KUKA KRL program: MyProgram_342().src

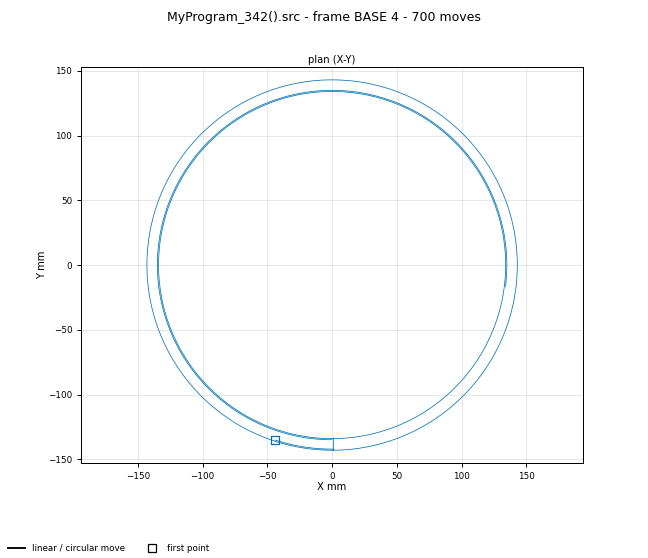
[picture p0: tool path of MyProgram_342().src in frame BASE 4, 700 of 700 moves have a stored position in this frame; points joined in program order, loops and branches not executed]
&ACCESS RVP
&REL 1
&PARAM TEMPLATE = C:\KRC\Roboter\Template\vorgabe
&PARAM EDITMASK = *
DEF MyProgram_342()
; ---- Setting reference (Base) ----
$BASE = BASE_DATA[4]

; --------------------------
; ---- Setting tool (TCP) ----
$TOOL = TOOL_DATA[3]
; --------------------------

$VEL.CP = VEL_APROX_PRINT
Startdeposition()
$VEL.CP = VEL_PRINT
LIN {X -44.0443,Y -135.0812,Z 191,A -94.9972,B 0.9183,C 0.2037,E1 0.9053,E2 187.7978} C_DIS
LIN {X -40.4187,Y -136.2083,Z 191,A -93.5168,B 0.9182,C 0.2043,E1 0.9093,E2 186.3246} C_DIS
LIN {X -37.0832,Y -137.1539,Z 191,A -92.1234,B 0.9181,C 0.2047,E1 0.9131,E2 184.9314} C_DIS
LIN {X -34.1943,Y -137.9034,Z 191,A -90.8718,B 0.9181,C 0.2049,E1 0.9166,E2 183.672} C_DIS
LIN {X -30.5962,Y -138.7458,Z 191,A -89.5644,B 0.9179,C 0.2055,E1 0.9201,E2 182.392} C_DIS
LIN {X -27.1259,Y -139.4652,Z 191,A -87.9953,B 0.9179,C 0.2052,E1 0.9245,E2 180.801} C_DIS
LIN {X -23.7617,Y -140.0774,Z 191,A -86.7669,B 0.9179,C 0.2056,E1 0.9279,E2 179.5949} C_DIS
LIN {X -20.9391,Y -140.5289,Z 191,A -85.3937,B 0.918,C 0.205,E1 0.9318,E2 178.1876} C_DIS
LIN {X -16.902,Y -141.0692,Z 191,A -84.0993,B 0.9178,C 0.2057,E1 0.9353,E2 176.9455} C_DIS
LIN {X -14.3962,Y -141.3492,Z 191,A -82.7514,B 0.9181,C 0.2046,E1 0.9393,E2 175.5466} C_DIS
LIN {X -10.0552,Y -141.7222,Z 191,A -81.1558,B 0.9181,C 0.2046,E1 0.9437,E2 173.9748} C_DIS
LIN {X -6.754,Y -141.9181,Z 191,A -79.8698,B 0.9181,C 0.2043,E1 0.9473,E2 172.6955} C_DIS
LIN {X -3.1252,Y -142.0459,Z 191,A -78.3714,B 0.9183,C 0.2036,E1 0.9516,E2 171.191} C_DIS
LIN {X 0.5232,Y -142.0775,Z 191,A -76.8992,B 0.9185,C 0.2029,E1 0.9557,E2 169.7179} C_DIS
LIN {X 0.5232,Y -142.0775,Z 191,A -76.8992,B 0.9185,C 0.2029,E1 0.9557,E2 169.7179} C_DIS
Enddeposition()
LIN {X 1.0243,Y -142.9726,Z 191,A -77.066,B 0.9181,C 0.2043,E1 0.955,E2 169.9648} C_DIS
Startdeposition()
$VEL.CP = VEL_PRINT
LIN {X -1.7511,Y -142.9678,Z 191,A -78.3434,B 0.9179,C 0.2053,E1 0.9513,E2 171.2682} C_DIS
LIN {X -5.1484,Y -142.885,Z 191,A -79.7715,B 0.9177,C 0.2061,E1 0.9473,E2 172.7072} C_DIS
LIN {X -8.6494,Y -142.7153,Z 191,A -81.1441,B 0.9177,C 0.2064,E1 0.9434,E2 174.0755} C_DIS
LIN {X -12.1449,Y -142.4604,Z 191,A -82.5233,B 0.9176,C 0.2067,E1 0.9395,E2 175.4516} C_DIS
LIN {X -15.6335,Y -142.1201,Z 191,A -83.9093,B 0.9176,C 0.2069,E1 0.9356,E2 176.8354} C_DIS
LIN {X -19.1308,Y -141.6924,Z 191,A -85.3144,B 0.9175,C 0.2071,E1 0.9316,E2 178.2402} C_DIS
LIN {X -22.712,Y -141.1639,Z 191,A -86.7484,B 0.9175,C 0.2071,E1 0.9276,E2 179.6723} C_DIS
LIN {X -25.7644,Y -140.6376,Z 191,A -88.0735,B 0.9175,C 0.2073,E1 0.9239,E2 181.0107} C_DIS
LIN {X -29.4674,Y -139.9092,Z 191,A -89.5418,B 0.9175,C 0.2071,E1 0.9198,E2 182.4729} C_DIS
LIN {X -33.0283,Y -139.1105,Z 191,A -90.9656,B 0.9175,C 0.2068,E1 0.9159,E2 183.8914} C_DIS
LIN {X -36.4402,Y -138.2557,Z 191,A -92.3295,B 0.9177,C 0.2064,E1 0.9122,E2 185.2488} C_DIS
LIN {X -39.8092,Y -137.3234,Z 191,A -93.8498,B 0.9177,C 0.2063,E1 0.908,E2 186.7878} C_DIS
LIN {X -43.0482,Y -136.343,Z 191,A -95.202,B 0.9177,C 0.2058,E1 0.9043,E2 188.14} C_DIS
LIN {X -46.4782,Y -135.2119,Z 191,A -96.7128,B 0.9179,C 0.2053,E1 0.9003,E2 189.6609} C_DIS
LIN {X -49.0096,Y -134.3156,Z 191,A -97.9561,B 0.9179,C 0.2051,E1 0.8969,E2 190.9301} C_DIS
LIN {X -53.0946,Y -132.7533,Z 191,A -99.6242,B 0.9182,C 0.2039,E1 0.8925,E2 192.5858} C_DIS
LIN {X -56.2262,Y -131.4582,Z 191,A -101.0289,B 0.9184,C 0.2032,E1 0.8888,E2 193.998} C_DIS
LIN {X -58.6861,Y -130.3778,Z 191,A -102.1543,B 0.9185,C 0.2025,E1 0.8859,E2 195.131} C_DIS
LIN {X -61.8637,Y -128.9001,Z 191,A -103.6197,B 0.9187,C 0.2015,E1 0.8821,E2 196.6061} C_DIS
LIN {X -65.0103,Y -127.342,Z 191,A -105.099,B 0.919,C 0.2005,E1 0.8783,E2 198.0966} C_DIS
LIN {X -68.3884,Y -125.5624,Z 191,A -106.7802,B 0.9192,C 0.1993,E1 0.8741,E2 199.8012} C_DIS
LIN {X -72.0014,Y -123.5268,Z 191,A -108.4575,B 0.9196,C 0.1977,E1 0.87,E2 201.481} C_DIS
LIN {X -74.9587,Y -121.7544,Z 191,A -109.9364,B 0.9198,C 0.1964,E1 0.8664,E2 202.9748} C_DIS
LIN {X -78.5539,Y -119.4662,Z 191,A -111.7694,B 0.9202,C 0.1947,E1 0.862,E2 204.8271} C_DIS
LIN {X -82.1648,Y -117.0125,Z 191,A -113.6368,B 0.9206,C 0.1927,E1 0.8576,E2 206.7124} C_DIS
LIN {X -85.116,Y -114.8837,Z 191,A -115.2771,B 0.921,C 0.191,E1 0.8538,E2 208.3803} C_DIS
LIN {X -88.608,Y -112.2125,Z 191,A -117.0907,B 0.9215,C 0.1887,E1 0.8497,E2 210.2018} C_DIS
LIN {X -91.5174,Y -109.8528,Z 191,A -118.854,B 0.9219,C 0.1867,E1 0.8458,E2 212.0045} C_DIS
LIN {X -94.7125,Y -107.1094,Z 191,A -120.5293,B 0.9224,C 0.1842,E1 0.8422,E2 213.6779} C_DIS
LIN {X -97.2632,Y -104.7989,Z 191,A -122.0448,B 0.9228,C 0.1821,E1 0.839,E2 215.2137} C_DIS
LIN {X -99.8004,Y -102.3863,Z 191,A -123.6022,B 0.9232,C 0.1799,E1 0.8358,E2 216.7943} C_DIS
LIN {X -102.7691,Y -99.4052,Z 191,A -125.495,B 0.9237,C 0.1771,E1 0.832,E2 218.7178} C_DIS
LIN {X -105.3467,Y -96.6693,Z 191,A -127.1186,B 0.9242,C 0.1745,E1 0.8289,E2 220.3587} C_DIS
LIN {X -108.0416,Y -93.6488,Z 191,A -128.8309,B 0.9248,C 0.1716,E1 0.8257,E2 222.0841} C_DIS
LIN {X -110.0019,Y -91.3373,Z 191,A -130.4103,B 0.9252,C 0.1694,E1 0.8227,E2 223.7174} C_DIS
LIN {X -112.7081,Y -87.977,Z 191,A -132.2096,B 0.9258,C 0.166,E1 0.8195,E2 225.5268} C_DIS
LIN {X -114.8262,Y -85.1932,Z 191,A -133.7873,B 0.9263,C 0.1632,E1 0.8168,E2 227.1302} C_DIS
LIN {X -116.9319,Y -82.2791,Z 191,A -135.5615,B 0.9268,C 0.1603,E1 0.8139,E2 228.9531} C_DIS
LIN {X -119.3971,Y -78.6588,Z 191,A -137.5331,B 0.9275,C 0.1565,E1 0.8107,E2 230.9559} C_DIS
LIN {X -121.6959,Y -75.054,Z 191,A -139.3334,B 0.9281,C 0.1528,E1 0.808,E2 232.7685} C_DIS
LIN {X -123.5289,Y -71.9976,Z 191,A -140.96,B 0.9286,C 0.1496,E1 0.8057,E2 234.4237} C_DIS
LIN {X -125.2281,Y -68.9993,Z 191,A -142.5485,B 0.9291,C 0.1464,E1 0.8034,E2 236.0418} C_DIS
LIN {X -126.8799,Y -65.9105,Z 191,A -144.1657,B 0.9296,C 0.143,E1 0.8013,E2 237.6895} C_DIS
LIN {X -128.4908,Y -62.7119,Z 191,A -145.7864,B 0.9302,C 0.1396,E1 0.7992,E2 239.3365} C_DIS
LIN {X -129.9345,Y -59.6614,Z 191,A -147.3777,B 0.9307,C 0.1362,E1 0.7973,E2 240.9617} C_DIS
LIN {X -131.3976,Y -56.3662,Z 191,A -148.9997,B 0.9312,C 0.1326,E1 0.7955,E2 242.6086} C_DIS
LIN {X -132.7118,Y -53.1975,Z 191,A -150.6229,B 0.9317,C 0.129,E1 0.7937,E2 244.2667} C_DIS
LIN {X -133.9822,Y -49.9116,Z 191,A -152.2574,B 0.9322,C 0.1254,E1 0.792,E2 245.9323} C_DIS
LIN {X -135.1575,Y -46.6351,Z 191,A -153.8995,B 0.9327,C 0.1216,E1 0.7905,E2 247.609} C_DIS
LIN {X -136.3021,Y -43.1765,Z 191,A -155.5832,B 0.9332,C 0.1177,E1 0.789,E2 249.3237} C_DIS
LIN {X -137.2869,Y -39.934,Z 191,A -157.1687,B 0.9336,C 0.114,E1 0.7877,E2 250.9407} C_DIS
LIN {X -138.2248,Y -36.5561,Z 191,A -158.8107,B 0.9341,C 0.1101,E1 0.7865,E2 252.6153} C_DIS
LIN {X -139.0565,Y -33.2525,Z 191,A -160.4242,B 0.9346,C 0.1063,E1 0.7854,E2 254.2629} C_DIS
LIN {X -139.7677,Y -30.1225,Z 191,A -161.9849,B 0.935,C 0.1026,E1 0.7844,E2 255.8611} C_DIS
LIN {X -140.5458,Y -26.2607,Z 191,A -163.7723,B 0.9354,C 0.0982,E1 0.7835,E2 257.6767} C_DIS
LIN {X -141.1657,Y -22.7011,Z 191,A -165.4595,B 0.9359,C 0.094,E1 0.7827,E2 259.3961} C_DIS
LIN {X -141.663,Y -19.355,Z 191,A -167.1313,B 0.9363,C 0.09,E1 0.782,E2 261.1107} C_DIS
LIN {X -142.1054,Y -15.7707,Z 191,A -168.7912,B 0.9367,C 0.0858,E1 0.7814,E2 262.7989} C_DIS
LIN {X -142.4479,Y -12.292,Z 191,A -170.4387,B 0.937,C 0.0817,E1 0.781,E2 264.4792} C_DIS
LIN {X -142.7058,Y -8.8037,Z 191,A -172.087,B 0.9374,C 0.0776,E1 0.7807,E2 266.1602} C_DIS
LIN {X -142.8807,Y -5.2595,Z 191,A -173.7528,B 0.9377,C 0.0734,E1 0.7805,E2 267.8582} C_DIS
LIN {X -142.9677,Y -1.7607,Z 191,A -175.3545,B 0.938,C 0.0693,E1 0.7804,E2 269.4859} C_DIS
LIN {X -142.9703,Y 1.6027,Z 191,A -177.0572,B 0.9383,C 0.0652,E1 0.7804,E2 271.2353} C_DIS
LIN {X -142.8852,Y 5.1432,Z 191,A -178.7056,B 0.9386,C 0.061,E1 0.7806,E2 272.9134} C_DIS
LIN {X -142.7147,Y 8.659,Z 191,A 179.6384,B 0.9389,C 0.0568,E1 0.7808,E2 274.601} C_DIS
LIN {X -142.46,Y 12.1493,Z 191,A 177.9898,B 0.9391,C 0.0527,E1 0.7812,E2 276.2813} C_DIS
LIN {X -142.1202,Y 15.6329,Z 191,A 176.3393,B 0.9393,C 0.0485,E1 0.7817,E2 277.9634} C_DIS
LIN {X -141.6952,Y 19.1092,Z 191,A 174.6795,B 0.9395,C 0.0444,E1 0.7823,E2 279.6559} C_DIS
LIN {X -141.1673,Y 22.6907,Z 191,A 172.9828,B 0.9397,C 0.0402,E1 0.783,E2 281.3838} C_DIS
LIN {X -140.6491,Y 25.7,Z 191,A 171.4402,B 0.9399,C 0.0365,E1 0.7838,E2 282.9668} C_DIS
LIN {X -139.885,Y 29.5794,Z 191,A 169.6984,B 0.94,C 0.0321,E1 0.7848,E2 284.728} C_DIS
LIN {X -139.1218,Y 32.9815,Z 191,A 168.0174,B 0.9402,C 0.028,E1 0.7858,E2 286.4445} C_DIS
LIN {X -138.2739,Y 36.3721,Z 191,A 166.375,B 0.9402,C 0.0241,E1 0.787,E2 288.1168} C_DIS
LIN {X -137.3203,Y 39.8199,Z 191,A 164.6972,B 0.9404,C 0.02,E1 0.7883,E2 289.8246} C_DIS
LIN {X -136.3377,Y 43.0651,Z 191,A 163.1033,B 0.9404,C 0.0163,E1 0.7896,E2 291.4473} C_DIS
LIN {X -135.1967,Y 46.5221,Z 191,A 161.409,B 0.9404,C 0.0123,E1 0.7912,E2 293.1703} C_DIS
LIN {X -134.0172,Y 49.818,Z 191,A 159.8681,B 0.9405,C 0.0086,E1 0.7927,E2 294.7277} C_DIS
LIN {X -132.7576,Y 53.084,Z 191,A 158.1472,B 0.9405,C 0.0048,E1 0.7945,E2 296.4873} C_DIS
LIN {X -131.2219,Y 56.7725,Z 191,A 156.2286,B 0.9405,C 0.0005,E1 0.7966,E2 298.444} C_DIS
LIN {X -129.6557,Y 60.2643,Z 191,A 154.5046,B 0.9405,C -0.0034,E1 0.7986,E2 300.1906} C_DIS
LIN {X -127.8296,Y 64.0521,Z 191,A 152.5628,B 0.9405,C -0.0076,E1 0.8011,E2 302.1629} C_DIS
LIN {X -126.0944,Y 67.4031,Z 191,A 150.8798,B 0.9405,C -0.0113,E1 0.8033,E2 303.8657} C_DIS
LIN {X -124.3943,Y 70.4918,Z 191,A 149.217,B 0.9405,C -0.0147,E1 0.8056,E2 305.5579} C_DIS
LIN {X -122.6024,Y 73.5643,Z 191,A 147.4166,B 0.9405,C -0.0181,E1 0.8082,E2 307.4027} C_DIS
LIN {X -120.326,Y 77.2305,Z 191,A 145.6237,B 0.9403,C -0.022,E1 0.8109,E2 309.2021} C_DIS
LIN {X -118.3683,Y 80.1987,Z 191,A 143.8437,B 0.9403,C -0.0252,E1 0.8138,E2 311.0236} C_DIS
LIN {X -115.9267,Y 83.6896,Z 191,A 142.0724,B 0.9401,C -0.0288,E1 0.8167,E2 312.8014} C_DIS
LIN {X -113.8414,Y 86.5056,Z 191,A 140.4645,B 0.9401,C -0.0318,E1 0.8194,E2 314.4326} C_DIS
LIN {X -111.5941,Y 89.3859,Z 191,A 138.6711,B 0.9399,C -0.0348,E1 0.8226,E2 316.2639} C_DIS
LIN {X -108.8784,Y 92.6735,Z 191,A 136.9142,B 0.9399,C -0.0381,E1 0.8258,E2 318.0253} C_DIS
LIN {X -106.5362,Y 95.3567,Z 191,A 135.2388,B 0.9397,C -0.0408,E1 0.829,E2 319.7288} C_DIS
LIN {X -103.5904,Y 98.5495,Z 191,A 133.4117,B 0.9396,C -0.0439,E1 0.8325,E2 321.5649} C_DIS
LIN {X -101.103,Y 101.1002,Z 191,A 131.6927,B 0.9394,C -0.0463,E1 0.836,E2 323.3169} C_DIS
LIN {X -97.9581,Y 104.1496,Z 191,A 129.8889,B 0.9393,C -0.0492,E1 0.8397,E2 325.1251} C_DIS
LIN {X -95.3755,Y 106.5195,Z 191,A 128.362,B 0.9392,C -0.0515,E1 0.8429,E2 326.6653} C_DIS
LIN {X -92.7655,Y 108.8002,Z 191,A 126.8125,B 0.9391,C -0.0536,E1 0.8462,E2 328.2323} C_DIS
LIN {X -89.3893,Y 111.5913,Z 191,A 124.9162,B 0.9389,C -0.0561,E1 0.8504,E2 330.1438} C_DIS
LIN {X -86.6273,Y 113.7483,Z 191,A 123.3944,B 0.9388,C -0.058,E1 0.8538,E2 331.6782} C_DIS
LIN {X -83.7666,Y 115.8709,Z 191,A 121.8524,B 0.9387,C -0.0598,E1 0.8574,E2 333.2323} C_DIS
LIN {X -80.2081,Y 118.3619,Z 191,A 120.0024,B 0.9385,C -0.0619,E1 0.8617,E2 335.0937} C_DIS
LIN {X -77.2858,Y 120.2907,Z 191,A 118.4769,B 0.9385,C -0.0634,E1 0.8654,E2 336.6323} C_DIS
LIN {X -73.5668,Y 122.6009,Z 191,A 116.6243,B 0.9383,C -0.0653,E1 0.8699,E2 338.4949} C_DIS
LIN {X -70.5413,Y 124.3661,Z 191,A 115.1433,B 0.9383,C -0.0666,E1 0.8735,E2 339.9839} C_DIS
LIN {X -67.4728,Y 126.0569,Z 191,A 113.6366,B 0.9381,C -0.0679,E1 0.8773,E2 341.5014} C_DIS
LIN {X -64.275,Y 127.7163,Z 191,A 112.1606,B 0.9381,C -0.0691,E1 0.881,E2 342.9801} C_DIS
LIN {X -61.0358,Y 129.2957,Z 191,A 110.5945,B 0.938,C -0.0701,E1 0.885,E2 344.5592} C_DIS
LIN {X -57.9783,Y 130.6944,Z 191,A 109.2192,B 0.9379,C -0.0711,E1 0.8886,E2 345.9368} C_DIS
LIN {X -53.9096,Y 132.4247,Z 191,A 107.2414,B 0.9379,C -0.072,E1 0.8938,E2 347.9367} C_DIS
LIN {X -49.8217,Y 134.0159,Z 191,A 105.5972,B 0.9377,C -0.0731,E1 0.8981,E2 349.5673} C_DIS
LIN {X -46.631,Y 135.1589,Z 191,A 104.1885,B 0.9377,C -0.0737,E1 0.9019,E2 350.981} C_DIS
LIN {X -43.0836,Y 136.3318,Z 191,A 102.5157,B 0.9377,C -0.0741,E1 0.9065,E2 352.6725} C_DIS
LIN {X -38.2252,Y 137.7725,Z 191,A 100.5903,B 0.9376,C -0.0749,E1 0.9117,E2 354.5852} C_DIS
LIN {X -34.3164,Y 138.8,Z 191,A 98.8052,B 0.9376,C -0.075,E1 0.9166,E2 356.388} C_DIS
LIN {X -30.2002,Y 139.751,Z 191,A 97.1875,B 0.9376,C -0.0754,E1 0.9211,E2 357.9965} C_DIS
LIN {X -26.2866,Y 140.5409,Z 191,A 95.6367,B 0.9376,C -0.0756,E1 0.9254,E2 359.5411} C_DIS
LIN {X -22.7225,Y 141.1622,Z 191,A 94.1997,B 0.9376,C -0.0756,E1 0.9294,E2 360.9762} C_DIS
LIN {X -19.3708,Y 141.661,Z 191,A 92.7853,B 0.9376,C -0.0754,E1 0.9334,E2 362.3962} C_DIS
LIN {X -15.7841,Y 142.1039,Z 191,A 91.5335,B 0.9376,C -0.0756,E1 0.9368,E2 363.6255} C_DIS
LIN {X -12.2682,Y 142.4499,Z 191,A 89.9925,B 0.9376,C -0.075,E1 0.9412,E2 365.1799} C_DIS
LIN {X -8.7735,Y 142.7077,Z 191,A 88.6162,B 0.9376,C -0.0747,E1 0.9451,E2 366.5524} C_DIS
LIN {X -5.6927,Y 142.8638,Z 191,A 87.3417,B 0.9376,C -0.0742,E1 0.9487,E2 367.8307} C_DIS
LIN {X -1.7582,Y 142.9677,Z 191,A 85.8854,B 0.9376,C -0.0738,E1 0.9528,E2 369.273} C_DIS
LIN {X 1.7562,Y 142.9677,Z 191,A 84.4997,B 0.9377,C -0.0732,E1 0.9567,E2 370.6556} C_DIS
LIN {X 5.1446,Y 142.8852,Z 191,A 83.1564,B 0.9377,C -0.0725,E1 0.9605,E2 371.9968} C_DIS
LIN {X 8.6439,Y 142.7156,Z 191,A 81.8057,B 0.9378,C -0.0717,E1 0.9643,E2 373.341} C_DIS
LIN {X 12.1399,Y 142.4608,Z 191,A 80.4574,B 0.9378,C -0.0709,E1 0.9681,E2 374.6825} C_DIS
LIN {X 15.4004,Y 142.1452,Z 191,A 79.1661,B 0.938,C -0.07,E1 0.9717,E2 375.9709} C_DIS
LIN {X 19.1264,Y 141.693,Z 191,A 77.756,B 0.938,C -0.0691,E1 0.9756,E2 377.3701} C_DIS
LIN {X 22.3424,Y 141.2213,Z 191,A 76.4997,B 0.9381,C -0.0681,E1 0.9791,E2 378.6208} C_DIS
LIN {X 26.0479,Y 140.5865,Z 191,A 75.0289,B 0.9382,C -0.0668,E1 0.9832,E2 380.0872} C_DIS
LIN {X 29.6046,Y 139.8795,Z 191,A 73.7235,B 0.9382,C -0.0658,E1 0.9868,E2 381.3754} C_DIS
LIN {X 33.0376,Y 139.1083,Z 191,A 72.3827,B 0.9384,C -0.0645,E1 0.9905,E2 382.708} C_DIS
LIN {X 36.4272,Y 138.2592,Z 191,A 71.0407,B 0.9384,C -0.0631,E1 0.9941,E2 384.043} C_DIS
LIN {X 39.7961,Y 137.3273,Z 191,A 69.7337,B 0.9385,C -0.0617,E1 0.9977,E2 385.3391} C_DIS
LIN {X 43.0376,Y 136.3464,Z 191,A 68.4532,B 0.9386,C -0.0603,E1 1.0011,E2 386.6106} C_DIS
LIN {X 45.7652,Y 135.4558,Z 191,A 67.2302,B 0.9387,C -0.0586,E1 1.0044,E2 387.8417} C_DIS
LIN {X 49.8206,Y 134.0163,Z 191,A 65.801,B 0.9388,C -0.0573,E1 1.0081,E2 389.2368} C_DIS
LIN {X 53.0912,Y 132.7546,Z 191,A 64.4671,B 0.9389,C -0.0556,E1 1.0116,E2 390.5623} C_DIS
LIN {X 56.2234,Y 131.4594,Z 191,A 63.2099,B 0.939,C -0.0539,E1 1.0148,E2 391.8077} C_DIS
LIN {X 59.481,Y 130.0179,Z 191,A 61.8734,B 0.9391,C -0.0521,E1 1.0182,E2 393.1335} C_DIS
LIN {X 62.7074,Y 128.493,Z 191,A 60.5917,B 0.9392,C -0.0504,E1 1.0214,E2 394.3979} C_DIS
LIN {X 65.785,Y 126.9458,Z 191,A 59.3322,B 0.9393,C -0.0486,E1 1.0246,E2 395.6431} C_DIS
LIN {X 68.8971,Y 125.2847,Z 191,A 57.993,B 0.9394,C -0.0466,E1 1.0279,E2 396.9736} C_DIS
LIN {X 72.5064,Y 123.2304,Z 191,A 56.3957,B 0.9395,C -0.0439,E1 1.0317,E2 398.5629} C_DIS
LIN {X 76.0974,Y 121.046,Z 191,A 54.8634,B 0.9397,C -0.0415,E1 1.0354,E2 400.0774} C_DIS
LIN {X 79.4847,Y 118.849,Z 191,A 53.3483,B 0.9397,C -0.039,E1 1.0389,E2 401.5803} C_DIS
LIN {X 83.0062,Y 116.4169,Z 191,A 51.9221,B 0.9399,C -0.0369,E1 1.0421,E2 402.9724} C_DIS
LIN {X 85.8738,Y 114.3183,Z 191,A 50.5144,B 0.9399,C -0.0342,E1 1.0453,E2 404.3782} C_DIS
LIN {X 89.3933,Y 111.5881,Z 191,A 48.8798,B 0.9401,C -0.0313,E1 1.0489,E2 405.995} C_DIS
LIN {X 93.1207,Y 108.4964,Z 191,A 47.2025,B 0.9401,C -0.0284,E1 1.0524,E2 407.641} C_DIS
LIN {X 96.5087,Y 105.4944,Z 191,A 45.607,B 0.9402,C -0.0255,E1 1.0557,E2 409.2104} C_DIS
LIN {X 99.1712,Y 102.9957,Z 191,A 44.2678,B 0.9402,C -0.0229,E1 1.0584,E2 410.5349} C_DIS
LIN {X 102.293,Y 99.8955,Z 191,A 42.7319,B 0.9404,C -0.0201,E1 1.0614,E2 412.0435} C_DIS
LIN {X 104.7507,Y 97.3149,Z 191,A 41.4555,B 0.9404,C -0.0176,E1 1.0638,E2 413.3016} C_DIS
LIN {X 107.6524,Y 94.0949,Z 191,A 39.922,B 0.9404,C -0.0145,E1 1.0666,E2 414.8105} C_DIS
LIN {X 109.9618,Y 91.3857,Z 191,A 38.6546,B 0.9405,C -0.012,E1 1.0689,E2 416.0588} C_DIS
LIN {X 112.1609,Y 88.6737,Z 191,A 37.4046,B 0.9405,C -0.0094,E1 1.071,E2 417.2906} C_DIS
LIN {X 114.4124,Y 85.7489,Z 191,A 35.9709,B 0.9405,C -0.0061,E1 1.0734,E2 418.7191} C_DIS
LIN {X 116.9333,Y 82.2771,Z 191,A 34.4626,B 0.9405,C -0.0029,E1 1.0759,E2 420.2017} C_DIS
LIN {X 119.3312,Y 78.7589,Z 191,A 33.0648,B 0.9405,C -0.0002,E1 1.078,E2 421.5616} C_DIS
LIN {X 121.2326,Y 75.8,Z 191,A 31.8082,B 0.9405,C 0.0025,E1 1.0798,E2 422.7994} C_DIS
LIN {X 123.0551,Y 72.8047,Z 191,A 30.5734,B 0.9405,C 0.0052,E1 1.0816,E2 424.0133} C_DIS
LIN {X 124.8026,Y 69.766,Z 191,A 29.2985,B 0.9405,C 0.0082,E1 1.0833,E2 425.2723} C_DIS
LIN {X 126.8917,Y 65.888,Z 191,A 27.7776,B 0.9405,C 0.0115,E1 1.0853,E2 426.7628} C_DIS
LIN {X 128.4917,Y 62.7099,Z 191,A 26.5378,B 0.9405,C 0.0142,E1 1.0868,E2 427.9796} C_DIS
LIN {X 129.9877,Y 59.5464,Z 191,A 25.2979,B 0.9405,C 0.0171,E1 1.0882,E2 429.1993} C_DIS
LIN {X 131.4128,Y 56.3311,Z 191,A 24.0622,B 0.9404,C 0.0199,E1 1.0896,E2 430.4133} C_DIS
LIN {X 132.7108,Y 53.2,Z 191,A 22.8726,B 0.9404,C 0.0227,E1 1.0908,E2 431.5818} C_DIS
LIN {X 134.015,Y 49.8239,Z 191,A 21.6139,B 0.9402,C 0.0255,E1 1.0921,E2 432.8164} C_DIS
LIN {X 134.9172,Y 47.3283,Z 191,A 20.5438,B 0.9402,C 0.0284,E1 1.0931,E2 433.8878} C_DIS
LIN {X 136.301,Y 43.18,Z 191,A 19.1789,B 0.9401,C 0.0312,E1 1.0942,E2 435.2034} C_DIS
LIN {X 137.2938,Y 39.9105,Z 191,A 17.9433,B 0.94,C 0.0342,E1 1.0952,E2 436.4222} C_DIS
LIN {X 138.228,Y 36.544,Z 191,A 16.7209,B 0.9398,C 0.0371,E1 1.096,E2 437.6221} C_DIS
LIN {X 139.012,Y 33.4371,Z 191,A 15.5654,B 0.9398,C 0.0399,E1 1.0968,E2 438.7613} C_DIS
LIN {X 139.8729,Y 29.6354,Z 191,A 14.2455,B 0.9396,C 0.043,E1 1.0976,E2 440.0502} C_DIS
LIN {X 140.5352,Y 26.3164,Z 191,A 13.0512,B 0.9395,C 0.0459,E1 1.0982,E2 441.2238} C_DIS
LIN {X 141.1642,Y 22.7099,Z 191,A 11.7836,B 0.9393,C 0.0489,E1 1.0988,E2 442.4658} C_DIS
LIN {X 141.6627,Y 19.3579,Z 191,A 10.5459,B 0.9391,C 0.052,E1 1.0993,E2 443.6883} C_DIS
LIN {X 142.1058,Y 15.7667,Z 191,A 9.3147,B 0.939,C 0.0549,E1 1.0996,E2 444.8911} C_DIS
LIN {X 142.4489,Y 12.281,Z 191,A 8.144,B 0.9388,C 0.0575,E1 1.0999,E2 446.0314} C_DIS
LIN {X 142.7083,Y 8.7626,Z 191,A 6.8692,B 0.9386,C 0.0607,E1 1.1002,E2 447.2884} C_DIS
LIN {X 142.8806,Y 5.2627,Z 191,A 5.6531,B 0.9384,C 0.0637,E1 1.1003,E2 448.48} C_DIS
LIN {X 142.9585,Y 2.3129,Z 191,A 4.5901,B 0.9382,C 0.0663,E1 1.1003,E2 449.5276} C_DIS
LIN {X 142.9701,Y -1.6151,Z 191,A 3.2153,B 0.938,C 0.0697,E1 1.1003,E2 450.8764} C_DIS
LIN {X 142.8849,Y -5.1529,Z 191,A 1.9953,B 0.9378,C 0.0726,E1 1.1003,E2 452.0703} C_DIS
LIN {X 142.715,Y -8.6539,Z 191,A 0.778,B 0.9375,C 0.0755,E1 1.1001,E2 453.263} C_DIS
LIN {X 142.46,Y -12.1495,Z 191,A -0.4413,B 0.9373,C 0.0784,E1 1.0998,E2 454.4578} C_DIS
LIN {X 142.1197,Y -15.6372,Z 191,A -1.6624,B 0.9371,C 0.0813,E1 1.0995,E2 455.6547} C_DIS
LIN {X 141.6942,Y -19.1171,Z 191,A -2.8916,B 0.9368,C 0.0843,E1 1.0991,E2 456.8607} C_DIS
LIN {X 141.163,Y -22.7174,Z 191,A -4.1511,B 0.9365,C 0.0872,E1 1.0985,E2 458.0937} C_DIS
LIN {X 140.5968,Y -25.9925,Z 191,A -5.3779,B 0.9362,C 0.0903,E1 1.0979,E2 459.3069} C_DIS
LIN {X 139.8798,Y -29.6033,Z 191,A -6.593,B 0.936,C 0.093,E1 1.0973,E2 460.4869} C_DIS
LIN {X 139.1125,Y -33.0202,Z 191,A -7.8473,B 0.9357,C 0.096,E1 1.0965,E2 461.7214} C_DIS
LIN {X 138.2616,Y -36.4181,Z 191,A -8.9799,B 0.9354,C 0.0984,E1 1.0957,E2 462.8171} C_DIS
LIN {X 137.6071,Y -38.8168,Z 191,A -9.9688,B 0.9351,C 0.1011,E1 1.095,E2 463.8057} C_DIS
LIN {X 136.3542,Y -43.0134,Z 191,A -11.4767,B 0.9348,C 0.1045,E1 1.0938,E2 465.2801} C_DIS
LIN {X 135.2002,Y -46.512,Z 191,A -12.7737,B 0.9344,C 0.1075,E1 1.0927,E2 466.5529} C_DIS
LIN {X 134.0175,Y -49.8172,Z 191,A -13.9785,B 0.9341,C 0.1102,E1 1.0915,E2 467.7302} C_DIS
LIN {X 132.7564,Y -53.0869,Z 191,A -15.2367,B 0.9338,C 0.1131,E1 1.0903,E2 468.9687} C_DIS
LIN {X 131.457,Y -56.2289,Z 191,A -16.4315,B 0.9334,C 0.1158,E1 1.089,E2 470.1408} C_DIS
LIN {X 130.3775,Y -58.6868,Z 191,A -17.4263,B 0.9331,C 0.1182,E1 1.0879,E2 471.1248} C_DIS
LIN {X 128.485,Y -62.7236,Z 191,A -18.9292,B 0.9327,C 0.1213,E1 1.0861,E2 472.5886} C_DIS
LIN {X 126.9432,Y -65.7898,Z 191,A -20.1626,B 0.9324,C 0.1241,E1 1.0846,E2 473.8028} C_DIS
LIN {X 125.2982,Y -68.8726,Z 191,A -21.4064,B 0.932,C 0.1269,E1 1.0829,E2 475.0252} C_DIS
LIN {X 123.5482,Y -71.9644,Z 191,A -22.6648,B 0.9316,C 0.1296,E1 1.0812,E2 476.2609} C_DIS
LIN {X 121.319,Y -75.6611,Z 191,A -24.2004,B 0.9311,C 0.1329,E1 1.079,E2 477.7698} C_DIS
LIN {X 119.4007,Y -78.6533,Z 191,A -25.463,B 0.9308,C 0.1355,E1 1.0771,E2 479.0102} C_DIS
LIN {X 116.9354,Y -82.2741,Z 191,A -26.9989,B 0.9303,C 0.1387,E1 1.0747,E2 480.5156} C_DIS
LIN {X 114.8835,Y -85.1163,Z 191,A -28.2437,B 0.9299,C 0.1412,E1 1.0727,E2 481.7383} C_DIS
LIN {X 112.7163,Y -87.9665,Z 191,A -29.5347,B 0.9295,C 0.1439,E1 1.0705,E2 483.0095} C_DIS
LIN {X 110.004,Y -91.3347,Z 191,A -31.0716,B 0.929,C 0.1469,E1 1.0679,E2 484.519} C_DIS
LIN {X 107.6936,Y -94.0477,Z 191,A -32.3437,B 0.9286,C 0.1494,E1 1.0656,E2 485.7695} C_DIS
LIN {X 105.275,Y -96.7474,Z 191,A -33.7452,B 0.9282,C 0.1524,E1 1.0629,E2 487.1646} C_DIS
LIN {X 102.3741,Y -99.8128,Z 191,A -35.1629,B 0.9278,C 0.1548,E1 1.0603,E2 488.5435} C_DIS
LIN {X 99.8956,Y -102.293,Z 191,A -36.4281,B 0.9274,C 0.1571,E1 1.0578,E2 489.7891} C_DIS
LIN {X 97.0984,Y -104.9523,Z 191,A -37.911,B 0.9269,C 0.1601,E1 1.0547,E2 491.2639} C_DIS
LIN {X 94.0924,Y -107.6546,Z 191,A -39.264,B 0.9265,C 0.1622,E1 1.052,E2 492.5786} C_DIS
LIN {X 91.38,Y -109.9665,Z 191,A -40.5511,B 0.9261,C 0.1644,E1 1.0493,E2 493.8459} C_DIS
LIN {X 88.6565,Y -112.1744,Z 191,A -41.9243,B 0.9256,C 0.1671,E1 1.0462,E2 495.2156} C_DIS
LIN {X 85.1765,Y -114.8386,Z 191,A -43.5101,B 0.9251,C 0.1697,E1 1.0427,E2 496.7773} C_DIS
LIN {X 81.5569,Y -117.4367,Z 191,A -45.1611,B 0.9246,C 0.1724,E1 1.039,E2 498.4097} C_DIS
LIN {X 77.9691,Y -119.8487,Z 191,A -46.6993,B 0.9242,C 0.1747,E1 1.0354,E2 499.9202} C_DIS
LIN {X 74.261,Y -122.1814,Z 191,A -48.2074,B 0.9238,C 0.1767,E1 1.0319,E2 501.3927} C_DIS
LIN {X 71.2935,Y -123.9366,Z 191,A -49.4957,B 0.9235,C 0.1787,E1 1.0288,E2 502.668} C_DIS
LIN {X 67.9845,Y -125.782,Z 191,A -51.003,B 0.923,C 0.1812,E1 1.0251,E2 504.1748} C_DIS
LIN {X 64.5997,Y -127.551,Z 191,A -52.3304,B 0.9227,C 0.1828,E1 1.0218,E2 505.4727} C_DIS
LIN {X 61.1456,Y -129.2432,Z 191,A -53.7225,B 0.9223,C 0.1845,E1 1.0183,E2 506.8436} C_DIS
LIN {X 57.9671,Y -130.6994,Z 191,A -55.0184,B 0.922,C 0.1862,E1 1.015,E2 508.1245} C_DIS
LIN {X 54.7518,Y -132.0784,Z 191,A -56.3109,B 0.9216,C 0.1878,E1 1.0117,E2 509.4016} C_DIS
LIN {X 51.9535,Y -133.2035,Z 191,A -57.5206,B 0.9213,C 0.1895,E1 1.0085,E2 510.6123} C_DIS
LIN {X 48.2794,Y -134.5789,Z 191,A -58.9092,B 0.921,C 0.1908,E1 1.0049,E2 511.9742} C_DIS
LIN {X 44.9654,Y -135.7221,Z 191,A -60.2404,B 0.9207,C 0.1924,E1 1.0014,E2 513.2952} C_DIS
LIN {X 41.4863,Y -136.8261,Z 191,A -61.5828,B 0.9204,C 0.1937,E1 0.9978,E2 514.6204} C_DIS
LIN {X 38.7988,Y -137.6121,Z 191,A -62.7442,B 0.9201,C 0.1951,E1 0.9947,E2 515.7886} C_DIS
LIN {X 34.8731,Y -138.659,Z 191,A -64.1851,B 0.9199,C 0.1963,E1 0.9908,E2 517.2021} C_DIS
LIN {X 31.4749,Y -139.4699,Z 191,A -65.5188,B 0.9196,C 0.1975,E1 0.9871,E2 518.5267} C_DIS
LIN {X 28.0523,Y -140.1987,Z 191,A -66.8389,B 0.9194,C 0.1986,E1 0.9835,E2 519.8352} C_DIS
LIN {X 24.444,Y -140.8739,Z 191,A -68.2351,B 0.9191,C 0.1997,E1 0.9797,E2 521.2209} C_DIS
LIN {X 21.0982,Y -141.4139,Z 191,A -69.5418,B 0.9189,C 0.2007,E1 0.976,E2 522.5206} C_DIS
LIN {X 17.5129,Y -141.9016,Z 191,A -70.9424,B 0.9187,C 0.2017,E1 0.9721,E2 523.9146} C_DIS
LIN {X 14.0313,Y -142.2874,Z 191,A -72.2887,B 0.9185,C 0.2026,E1 0.9683,E2 525.2529} C_DIS
LIN {X 10.5172,Y -142.5898,Z 191,A -73.6461,B 0.9183,C 0.2034,E1 0.9645,E2 526.6026} C_DIS
LIN {X 7.0188,Y -142.8048,Z 191,A -74.9982,B 0.9182,C 0.2041,E1 0.9607,E2 527.9475} C_DIS
LIN {X 3.5163,Y -142.9346,Z 191,A -76.3521,B 0.918,C 0.2047,E1 0.9569,E2 529.2944} C_DIS
LIN {X 1.0243,Y -142.9726,Z 191,A -77.0655,B 0.9181,C 0.2043,E1 0.955,E2 529.9646} C_DIS
Enddeposition()
LIN {X 0.9701,Y -133.9923,Z 192,A -63.8032,B 0.3093,C 0.1491,E1 0.38,E2 514.628} C_DIS
Startdeposition()
$VEL.CP = VEL_PRINT
LIN {X 0.9701,Y -133.9923,Z 192,A -63.8124,B 0.3093,C 0.1491,E1 0.3799,E2 514.6387} C_DIS
LIN {X 4.2382,Y -133.9322,Z 192,A -62.4464,B 0.3101,C 0.1473,E1 0.384,E2 513.2767} C_DIS
LIN {X 7.2635,Y -133.8022,Z 192,A -61.2247,B 0.3108,C 0.1458,E1 0.3877,E2 512.0654} C_DIS
LIN {X 11.4912,Y -133.5046,Z 192,A -59.8515,B 0.3114,C 0.1445,E1 0.3917,E2 510.7602} C_DIS
LIN {X 14.7548,Y -133.1839,Z 192,A -58.6981,B 0.3121,C 0.1431,E1 0.3951,E2 509.645} C_DIS
LIN {X 18.004,Y -132.7844,Z 192,A -57.5509,B 0.3127,C 0.1418,E1 0.3984,E2 508.5365} C_DIS
LIN {X 21.2355,Y -132.3067,Z 192,A -56.3887,B 0.3133,C 0.1403,E1 0.4018,E2 507.4101} C_DIS
LIN {X 24.5251,Y -131.736,Z 192,A -55.2361,B 0.314,C 0.1389,E1 0.4051,E2 506.2995} C_DIS
LIN {X 28.4108,Y -130.9515,Z 192,A -53.8473,B 0.3148,C 0.137,E1 0.4091,E2 504.9574} C_DIS
LIN {X 32.5482,Y -129.9855,Z 192,A -52.3092,B 0.3157,C 0.1348,E1 0.4135,E2 503.4615} C_DIS
LIN {X 36.396,Y -128.9607,Z 192,A -51.0554,B 0.3164,C 0.1332,E1 0.4169,E2 502.2765} C_DIS
LIN {X 39.5471,Y -128.0295,Z 192,A -49.9388,B 0.3171,C 0.1316,E1 0.42,E2 501.2038} C_DIS
LIN {X 42.6742,Y -127.0214,Z 192,A -48.7679,B 0.3178,C 0.1298,E1 0.4232,E2 500.0682} C_DIS
LIN {X 46.69,Y -125.6007,Z 192,A -47.3938,B 0.3186,C 0.1279,E1 0.4269,E2 498.7621} C_DIS
LIN {X 50.298,Y -124.1996,Z 192,A -46.0638,B 0.3194,C 0.1258,E1 0.4304,E2 497.4811} C_DIS
LIN {X 54.2758,Y -122.5142,Z 192,A -44.6593,B 0.3203,C 0.1236,E1 0.4341,E2 496.1437} C_DIS
LIN {X 57.2884,Y -121.135,Z 192,A -43.558,B 0.321,C 0.1218,E1 0.4369,E2 495.0899} C_DIS
LIN {X 60.2478,Y -119.691,Z 192,A -42.4692,B 0.3216,C 0.1201,E1 0.4397,E2 494.0491} C_DIS
LIN {X 63.7644,Y -117.8565,Z 192,A -41.1527,B 0.3225,C 0.1178,E1 0.4429,E2 492.7895} C_DIS
LIN {X 66.6585,Y -116.2439,Z 192,A -40.0322,B 0.3232,C 0.1159,E1 0.4457,E2 491.7132} C_DIS
LIN {X 70.2993,Y -114.0789,Z 192,A -38.5738,B 0.3241,C 0.1133,E1 0.4492,E2 490.3073} C_DIS
LIN {X 73.6417,Y -111.95,Z 192,A -37.3659,B 0.3248,C 0.1113,E1 0.452,E2 489.1722} C_DIS
LIN {X 76.3596,Y -110.1143,Z 192,A -36.327,B 0.3254,C 0.1094,E1 0.4544,E2 488.1873} C_DIS
LIN {X 79.2559,Y -108.0482,Z 192,A -35.0854,B 0.3262,C 0.107,E1 0.4572,E2 486.9868} C_DIS
LIN {X 82.8286,Y -105.3344,Z 192,A -33.6834,B 0.327,C 0.1045,E1 0.4603,E2 485.6613} C_DIS
LIN {X 85.9981,Y -102.7632,Z 192,A -32.327,B 0.3278,C 0.1019,E1 0.4632,E2 484.362} C_DIS
LIN {X 89.3367,Y -99.8742,Z 192,A -30.9511,B 0.3286,C 0.0994,E1 0.466,E2 483.0614} C_DIS
LIN {X 92.2828,Y -97.1595,Z 192,A -29.6202,B 0.3294,C 0.0967,E1 0.4687,E2 481.7861} C_DIS
LIN {X 95.3181,Y -94.1834,Z 192,A -28.2951,B 0.3302,C 0.0941,E1 0.4712,E2 480.5328} C_DIS
LIN {X 98.2489,Y -91.1216,Z 192,A -26.9071,B 0.3309,C 0.0913,E1 0.4738,E2 479.2062} C_DIS
LIN {X 101.2655,Y -87.7574,Z 192,A -25.4772,B 0.3317,C 0.0884,E1 0.4764,E2 477.8488} C_DIS
LIN {X 104.1055,Y -84.3685,Z 192,A -24.1242,B 0.3324,C 0.0858,E1 0.4787,E2 476.5731} C_DIS
LIN {X 106.6311,Y -81.153,Z 192,A -22.7927,B 0.3331,C 0.0829,E1 0.4809,E2 475.3011} C_DIS
LIN {X 109.1218,Y -77.7713,Z 192,A -21.4608,B 0.3338,C 0.0801,E1 0.483,E2 474.0352} C_DIS
LIN {X 111.4188,Y -74.4429,Z 192,A -20.2929,B 0.3344,C 0.0778,E1 0.4848,E2 472.9471} C_DIS
LIN {X 113.2096,Y -71.6905,Z 192,A -19.1816,B 0.3349,C 0.0753,E1 0.4864,E2 471.8769} C_DIS
LIN {X 115.2793,Y -68.3133,Z 192,A -17.9603,B 0.3355,C 0.0728,E1 0.4881,E2 470.7219} C_DIS
LIN {X 117.2987,Y -64.7838,Z 192,A -16.731,B 0.3361,C 0.0702,E1 0.4897,E2 469.5639} C_DIS
LIN {X 119.255,Y -61.1043,Z 192,A -15.4558,B 0.3366,C 0.0674,E1 0.4913,E2 468.3589} C_DIS
LIN {X 120.8414,Y -57.9028,Z 192,A -14.3963,B 0.3371,C 0.0652,E1 0.4925,E2 467.3642} C_DIS
LIN {X 122.1105,Y -55.1785,Z 192,A -13.4098,B 0.3375,C 0.0629,E1 0.4936,E2 466.4186} C_DIS
LIN {X 123.5068,Y -51.9768,Z 192,A -12.3654,B 0.3379,C 0.0607,E1 0.4947,E2 465.4358} C_DIS
LIN {X 124.7736,Y -48.8575,Z 192,A -11.2794,B 0.3383,C 0.0582,E1 0.4958,E2 464.3977} C_DIS
LIN {X 125.8368,Y -46.0532,Z 192,A -10.3508,B 0.3387,C 0.0561,E1 0.4967,E2 463.5171} C_DIS
LIN {X 127.014,Y -42.6965,Z 192,A -9.1568,B 0.3392,C 0.0532,E1 0.4977,E2 462.3669} C_DIS
LIN {X 128.2224,Y -38.9169,Z 192,A -8.0222,B 0.3395,C 0.0508,E1 0.4986,E2 461.3079} C_DIS
LIN {X 129.2155,Y -35.4848,Z 192,A -6.8107,B 0.34,C 0.0479,E1 0.4995,E2 460.1384} C_DIS
LIN {X 130.1467,Y -31.8991,Z 192,A -5.7682,B 0.3403,C 0.0456,E1 0.5002,E2 459.1678} C_DIS
LIN {X 130.9509,Y -28.4132,Z 192,A -4.6034,B 0.3406,C 0.0429,E1 0.5008,E2 458.0509} C_DIS
LIN {X 131.7359,Y -24.5261,Z 192,A -3.4143,B 0.341,C 0.0402,E1 0.5014,E2 456.9282} C_DIS
LIN {X 132.2982,Y -21.2897,Z 192,A -2.4347,B 0.3412,C 0.0379,E1 0.5019,E2 456.0039} C_DIS
LIN {X 132.7797,Y -18.0399,Z 192,A -1.3216,B 0.3415,C 0.0352,E1 0.5023,E2 454.9283} C_DIS
LIN {X 133.2835,Y -13.829,Z 192,A -0.1354,B 0.3418,C 0.0326,E1 0.5026,E2 453.8228} C_DIS
LIN {X 133.5695,Y -10.7239,Z 192,A 0.9019,B 0.342,C 0.0301,E1 0.5028,E2 452.823} C_DIS
LIN {X 133.8366,Y -6.5796,Z 192,A 2.1007,B 0.3422,C 0.0274,E1 0.503,E2 451.6974} C_DIS
LIN {X 133.9734,Y -2.6057,Z 192,A 3.3799,B 0.3425,C 0.0243,E1 0.5031,E2 450.471} C_DIS
LIN {X 133.9893,Y 1.6505,Z 192,A 4.6433,B 0.3426,C 0.0214,E1 0.5031,E2 449.277} C_DIS
LIN {X 133.9077,Y 4.9322,Z 192,A 5.6428,B 0.3428,C 0.019,E1 0.5031,E2 448.3275} C_DIS
LIN {X 133.7463,Y 8.2125,Z 192,A 6.6443,B 0.3429,C 0.0166,E1 0.5029,E2 447.3754} C_DIS
LIN {X 133.505,Y 11.4872,Z 192,A 7.6468,B 0.343,C 0.0143,E1 0.5027,E2 446.4219} C_DIS
LIN {X 133.184,Y 14.754,Z 192,A 8.6514,B 0.3431,C 0.0119,E1 0.5024,E2 445.4656} C_DIS
LIN {X 132.7226,Y 18.4508,Z 192,A 9.7183,B 0.3431,C 0.0095,E1 0.502,E2 444.4619} C_DIS
LIN {X 132.2455,Y 21.6055,Z 192,A 10.8369,B 0.3432,C 0.0066,E1 0.5015,E2 443.3725} C_DIS
LIN {X 131.6095,Y 25.1872,Z 192,A 11.8919,B 0.3432,C 0.0042,E1 0.501,E2 442.3768} C_DIS
LIN {X 130.9147,Y 28.5813,Z 192,A 12.9608,B 0.3433,C 0.0017,E1 0.5005,E2 441.3563} C_DIS
LIN {X 129.9825,Y 32.5598,Z 192,A 14.3022,B 0.3433,C -0.0016,E1 0.4996,E2 440.062} C_DIS
LIN {X 128.9611,Y 36.3946,Z 192,A 15.4244,B 0.3433,C -0.0041,E1 0.4988,E2 439.0062} C_DIS
LIN {X 127.8306,Y 40.1887,Z 192,A 16.6983,B 0.3433,C -0.0072,E1 0.4978,E2 437.7801} C_DIS
LIN {X 126.709,Y 43.5927,Z 192,A 17.7428,B 0.3432,C -0.0096,E1 0.4969,E2 436.7909} C_DIS
LIN {X 125.5984,Y 46.6961,Z 192,A 18.8431,B 0.3431,C -0.0123,E1 0.4959,E2 435.7252} C_DIS
LIN {X 123.9219,Y 50.9827,Z 192,A 20.2339,B 0.343,C -0.0155,E1 0.4945,E2 434.3987} C_DIS
LIN {X 122.3865,Y 54.5614,Z 192,A 21.308,B 0.3428,C -0.0178,E1 0.4934,E2 433.3896} C_DIS
LIN {X 121.1382,Y 57.2816,Z 192,A 22.326,B 0.3428,C -0.0203,E1 0.4922,E2 432.4001} C_DIS
LIN {X 119.6898,Y 60.2502,Z 192,A 23.302,B 0.3426,C -0.0225,E1 0.491,E2 431.4713} C_DIS
LIN {X 117.8536,Y 63.7699,Z 192,A 24.5356,B 0.3424,C -0.0254,E1 0.4895,E2 430.2874} C_DIS
LIN {X 116.2543,Y 66.6402,Z 192,A 25.5837,B 0.3422,C -0.0278,E1 0.488,E2 429.2771} C_DIS
LIN {X 114.0806,Y 70.2966,Z 192,A 26.9571,B 0.3419,C -0.031,E1 0.4861,E2 427.9504} C_DIS
LIN {X 111.9555,Y 73.6334,Z 192,A 28.0851,B 0.3417,C -0.0335,E1 0.4844,E2 426.8809} C_DIS
LIN {X 110.1236,Y 76.3462,Z 192,A 29.0972,B 0.3414,C -0.0358,E1 0.4829,E2 425.9087} C_DIS
LIN {X 108.0331,Y 79.2765,Z 192,A 30.3059,B 0.3411,C -0.0386,E1 0.4809,E2 424.7335} C_DIS
LIN {X 105.3428,Y 82.8178,Z 192,A 31.6441,B 0.3408,C -0.0415,E1 0.4787,E2 423.452} C_DIS
LIN {X 102.7495,Y 86.0143,Z 192,A 32.9702,B 0.3404,C -0.0445,E1 0.4763,E2 422.1691} C_DIS
LIN {X 99.839,Y 89.376,Z 192,A 34.3185,B 0.34,C -0.0474,E1 0.4739,E2 420.875} C_DIS
LIN {X 97.054,Y 92.3931,Z 192,A 35.6297,B 0.3396,C -0.0503,E1 0.4714,E2 419.6069} C_DIS
LIN {X 94.1689,Y 95.3324,Z 192,A 36.7449,B 0.3393,C -0.0525,E1 0.4693,E2 418.5536} C_DIS
LIN {X 92.0431,Y 97.3857,Z 192,A 37.8289,B 0.3389,C -0.055,E1 0.4671,E2 417.4865} C_DIS
LIN {X 89.0166,Y 100.1603,Z 192,A 39.1311,B 0.3384,C -0.0577,E1 0.4643,E2 416.2268} C_DIS
LIN {X 86.0126,Y 102.751,Z 192,A 40.3907,B 0.338,C -0.0603,E1 0.4617,E2 415.0076} C_DIS
LIN {X 82.5192,Y 105.5774,Z 192,A 41.7667,B 0.3375,C -0.0631,E1 0.4587,E2 413.6814} C_DIS
LIN {X 79.2733,Y 108.0355,Z 192,A 43.0818,B 0.3369,C -0.0658,E1 0.4557,E2 412.4046} C_DIS
LIN {X 75.8091,Y 110.4938,Z 192,A 44.4021,B 0.3364,C -0.0684,E1 0.4526,E2 411.1284} C_DIS
LIN {X 73.0763,Y 112.32,Z 192,A 45.4535,B 0.336,C -0.0705,E1 0.4501,E2 410.1081} C_DIS
LIN {X 69.7143,Y 114.4377,Z 192,A 46.733,B 0.3355,C -0.073,E1 0.447,E2 408.865} C_DIS
LIN {X 66.6565,Y 116.245,Z 192,A 47.9703,B 0.3349,C -0.0754,E1 0.444,E2 407.652} C_DIS
LIN {X 63.1912,Y 118.1645,Z 192,A 49.2802,B 0.3343,C -0.0779,E1 0.4406,E2 406.3747} C_DIS
LIN {X 59.6375,Y 119.9954,Z 192,A 50.5251,B 0.3338,C -0.0802,E1 0.4375,E2 405.1687} C_DIS
LIN {X 55.8018,Y 121.8268,Z 192,A 51.934,B 0.3332,C -0.0828,E1 0.4338,E2 403.7937} C_DIS
LIN {X 52.1619,Y 123.4295,Z 192,A 53.1334,B 0.3327,C -0.0848,E1 0.4306,E2 402.635} C_DIS
LIN {X 48.8667,Y 124.77,Z 192,A 54.4087,B 0.3321,C -0.0871,E1 0.4271,E2 401.3797} C_DIS
LIN {X 44.5233,Y 126.3864,Z 192,A 55.9023,B 0.3314,C -0.0896,E1 0.4231,E2 399.925} C_DIS
LIN {X 40.4889,Y 127.7347,Z 192,A 57.2546,B 0.3308,C -0.0918,E1 0.4193,E2 398.6091} C_DIS
LIN {X 37.3228,Y 128.6955,Z 192,A 58.3552,B 0.3303,C -0.0936,E1 0.4162,E2 397.5329} C_DIS
LIN {X 34.1489,Y 129.574,Z 192,A 59.5578,B 0.3297,C -0.0956,E1 0.4128,E2 396.3462} C_DIS
LIN {X 30.2982,Y 130.5285,Z 192,A 60.8571,B 0.3292,C -0.0975,E1 0.409,E2 395.077} C_DIS
LIN {X 26.8149,Y 131.2875,Z 192,A 62.0865,B 0.3286,C -0.0994,E1 0.4055,E2 393.8697} C_DIS
LIN {X 22.9105,Y 132.0267,Z 192,A 63.3523,B 0.3281,C -0.1012,E1 0.4018,E2 392.636} C_DIS
LIN {X 19.6582,Y 132.5501,Z 192,A 64.5022,B 0.3276,C -0.1028,E1 0.3984,E2 391.5051} C_DIS
LIN {X 16.404,Y 132.9913,Z 192,A 65.7283,B 0.327,C -0.1046,E1 0.3947,E2 390.292} C_DIS
LIN {X 12.1872,Y 133.4442,Z 192,A 67.0735,B 0.3265,C -0.1062,E1 0.3907,E2 388.9804} C_DIS
LIN {X 9.1941,Y 133.6835,Z 192,A 68.1915,B 0.326,C -0.1077,E1 0.3873,E2 387.8742} C_DIS
LIN {X 5.9196,Y 133.8692,Z 192,A 69.3246,B 0.3255,C -0.1091,E1 0.3839,E2 386.7602} C_DIS
LIN {X 2.6073,Y 133.9734,Z 192,A 70.4799,B 0.3251,C -0.1105,E1 0.3804,E2 385.623} C_DIS
LIN {X -1.6357,Y 133.9896,Z 192,A 72.0001,B 0.3245,C -0.1122,E1 0.3758,E2 384.1233} C_DIS
LIN {X -5.2256,Y 133.8963,Z 192,A 73.3162,B 0.324,C -0.1136,E1 0.3718,E2 382.8222} C_DIS
LIN {X -9.1634,Y 133.6858,Z 192,A 74.7208,B 0.3235,C -0.115,E1 0.3675,E2 381.4369} C_DIS
LIN {X -12.1757,Y 133.4453,Z 192,A 75.8188,B 0.3231,C -0.1161,E1 0.3642,E2 380.352} C_DIS
LIN {X -15.7171,Y 133.0732,Z 192,A 77.2074,B 0.3226,C -0.1174,E1 0.3599,E2 378.9725} C_DIS
LIN {X -19.6465,Y 132.5518,Z 192,A 78.5763,B 0.3222,C -0.1185,E1 0.3557,E2 377.6252} C_DIS
LIN {X -22.8861,Y 132.0311,Z 192,A 79.8961,B 0.3218,C -0.1196,E1 0.3517,E2 376.3113} C_DIS
LIN {X -26.8107,Y 131.2884,Z 192,A 81.3265,B 0.3214,C -0.1206,E1 0.3474,E2 374.8989} C_DIS
LIN {X -30.2909,Y 130.5301,Z 192,A 82.8141,B 0.321,C -0.1216,E1 0.3428,E2 373.4142} C_DIS
LIN {X -34.1446,Y 129.5752,Z 192,A 84.3485,B 0.3207,C -0.1226,E1 0.3382,E2 371.8906} C_DIS
LIN {X -37.978,Y 128.5037,Z 192,A 85.7738,B 0.3204,C -0.1233,E1 0.334,E2 370.483} C_DIS
LIN {X -41.118,Y 127.5337,Z 192,A 87.073,B 0.3202,C -0.1239,E1 0.3301,E2 369.1909} C_DIS
LIN {X -44.5127,Y 126.3901,Z 192,A 88.6531,B 0.3199,C -0.1246,E1 0.3254,E2 367.6085} C_DIS
LIN {X -48.8631,Y 124.7714,Z 192,A 90.4044,B 0.3197,C -0.1251,E1 0.3203,E2 365.8722} C_DIS
LIN {X -52.7905,Y 123.1613,Z 192,A 92.1117,B 0.3196,C -0.1255,E1 0.3153,E2 364.1721} C_DIS
LIN {X -55.7928,Y 121.8309,Z 192,A 93.5533,B 0.3195,C -0.1257,E1 0.3112,E2 362.7289} C_DIS
LIN {X -58.7614,Y 120.4275,Z 192,A 94.942,B 0.3195,C -0.1259,E1 0.3072,E2 361.3418} C_DIS
LIN {X -62.3162,Y 118.6257,Z 192,A 96.4668,B 0.3195,C -0.1259,E1 0.303,E2 359.8284} C_DIS
LIN {X -65.2233,Y 117.0553,Z 192,A 97.9835,B 0.3195,C -0.1259,E1 0.2988,E2 358.3062} C_DIS
LIN {X -68.3028,Y 115.2855,Z 192,A 99.6783,B 0.3195,C -0.1256,E1 0.2941,E2 356.6015} C_DIS
LIN {X -72.2469,Y 112.8552,Z 192,A 101.6372,B 0.3197,C -0.1252,E1 0.2889,E2 354.6448} C_DIS
LIN {X -75.0115,Y 111.0369,Z 192,A 103.0806,B 0.3198,C -0.1248,E1 0.2851,E2 353.2004} C_DIS
LIN {X -77.7099,Y 109.1658,Z 192,A 104.6562,B 0.3201,C -0.1242,E1 0.281,E2 351.6151} C_DIS
LIN {X -81.1459,Y 106.6366,Z 192,A 106.6892,B 0.3204,C -0.1233,E1 0.2759,E2 349.5701} C_DIS
LIN {X -84.3732,Y 104.1017,Z 192,A 108.6335,B 0.3208,C -0.1222,E1 0.2711,E2 347.6149} C_DIS
LIN {X -87.7789,Y 101.247,Z 192,A 110.794,B 0.3214,C -0.1208,E1 0.2659,E2 345.4391} C_DIS
LIN {X -90.8374,Y 98.5115,Z 192,A 112.7947,B 0.3219,C -0.1193,E1 0.2612,E2 343.4237} C_DIS
LIN {X -93.9299,Y 95.5673,Z 192,A 114.8963,B 0.3226,C -0.1175,E1 0.2565,E2 341.3053} C_DIS
LIN {X -96.8114,Y 92.647,Z 192,A 117.0162,B 0.3233,C -0.1155,E1 0.2518,E2 339.1626} C_DIS
LIN {X -99.6018,Y 89.6409,Z 192,A 119.1796,B 0.3241,C -0.1133,E1 0.2473,E2 336.9731} C_DIS
LIN {X -102.236,Y 86.6242,Z 192,A 121.3363,B 0.3249,C -0.1108,E1 0.2429,E2 334.7874} C_DIS
LIN {X -104.9189,Y 83.3543,Z 192,A 123.5996,B 0.3259,C -0.1081,E1 0.2384,E2 332.494} C_DIS
LIN {X -107.0502,Y 80.5989,Z 192,A 125.4675,B 0.3267,C -0.1056,E1 0.2349,E2 330.6006} C_DIS
LIN {X -109.3817,Y 77.4053,Z 192,A 127.7976,B 0.3277,C -0.1023,E1 0.2307,E2 328.226} C_DIS
LIN {X -111.4182,Y 74.4439,Z 192,A 129.7843,B 0.3286,C -0.0993,E1 0.2273,E2 326.2075} C_DIS
LIN {X -113.5107,Y 71.2134,Z 192,A 132.0836,B 0.3297,C -0.0957,E1 0.2234,E2 323.8609} C_DIS
LIN {X -115.5158,Y 67.9119,Z 192,A 134.5056,B 0.3308,C -0.0917,E1 0.2196,E2 321.3812} C_DIS
LIN {X -117.3924,Y 64.6146,Z 192,A 136.7129,B 0.3319,C -0.0878,E1 0.2163,E2 319.1293} C_DIS
LIN {X -119.2499,Y 61.1143,Z 192,A 139.2249,B 0.3331,C -0.0832,E1 0.2128,E2 316.553} C_DIS
LIN {X -121.168,Y 57.2194,Z 192,A 142.1664,B 0.3344,C -0.0775,E1 0.2089,E2 313.5234} C_DIS
LIN {X -121.168,Y 57.2194,Z 192,A 142.1649,B 0.3344,C -0.0775,E1 0.2089,E2 313.5249} C_DIS
LIN {X -122.7817,Y 53.6687,Z 192,A 144.497,B 0.3355,C -0.0728,E1 0.206,E2 311.1375} C_DIS
LIN {X -124.0603,Y 50.6436,Z 192,A 146.8095,B 0.3365,C -0.068,E1 0.2034,E2 308.747} C_DIS
LIN {X -124.0603,Y 50.6436,Z 192,A 146.8085,B 0.3365,C -0.068,E1 0.2034,E2 308.7481} C_DIS
LIN {X -125.3622,Y 47.3267,Z 192,A 148.9229,B 0.3374,C -0.0634,E1 0.2011,E2 306.582} C_DIS
LIN {X -126.393,Y 44.5043,Z 192,A 151.2766,B 0.3383,C -0.0582,E1 0.1987,E2 304.1319} C_DIS
LIN {X -126.393,Y 44.5043,Z 192,A 151.2753,B 0.3383,C -0.0582,E1 0.1987,E2 304.1334} C_DIS
LIN {X -127.7395,Y 40.4738,Z 192,A 154.0846,B 0.3394,C -0.0518,E1 0.1961,E2 301.232} C_DIS
LIN {X -127.7395,Y 40.4738,Z 192,A 154.0835,B 0.3394,C -0.0518,E1 0.1961,E2 301.2332} C_DIS
LIN {X -128.6935,Y 37.3298,Z 192,A 156.4591,B 0.3402,C -0.0463,E1 0.1941,E2 298.7649} C_DIS
LIN {X -128.6935,Y 37.3298,Z 192,A 156.4579,B 0.3402,C -0.0463,E1 0.1941,E2 298.7662} C_DIS
LIN {X -129.7965,Y 33.2929,Z 192,A 159.1693,B 0.341,C -0.0398,E1 0.192,E2 295.9649} C_DIS
LIN {X -129.7965,Y 33.2929,Z 192,A 159.1682,B 0.341,C -0.0398,E1 0.192,E2 295.9662} C_DIS
LIN {X -130.4648,Y 30.5769,Z 192,A 161.3681,B 0.3416,C -0.0345,E1 0.1905,E2 293.6654} C_DIS
LIN {X -130.4648,Y 30.5769,Z 192,A 161.3669,B 0.3416,C -0.0345,E1 0.1905,E2 293.6668} C_DIS
LIN {X -131.0943,Y 27.7492,Z 192,A 163.5116,B 0.3421,C -0.0292,E1 0.1891,E2 291.4288} C_DIS
LIN {X -131.0943,Y 27.7492,Z 192,A 163.5106,B 0.3421,C -0.0292,E1 0.1891,E2 291.43} C_DIS
LIN {X -131.7357,Y 24.5268,Z 192,A 166.0749,B 0.3426,C -0.0228,E1 0.1877,E2 288.7434} C_DIS
LIN {X -131.7357,Y 24.5268,Z 192,A 166.0731,B 0.3426,C -0.0228,E1 0.1877,E2 288.7454} C_DIS
LIN {X -132.2983,Y 21.289,Z 192,A 168.3978,B 0.3429,C -0.0169,E1 0.1866,E2 286.3215} C_DIS
LIN {X -132.2983,Y 21.289,Z 192,A 168.3964,B 0.3429,C -0.0169,E1 0.1866,E2 286.3231} C_DIS
LIN {X -132.8627,Y 17.4065,Z 192,A 171.3285,B 0.3432,C -0.0094,E1 0.1854,E2 283.2522} C_DIS
LIN {X -132.8627,Y 17.4065,Z 192,A 171.3266,B 0.3432,C -0.0094,E1 0.1854,E2 283.2542} C_DIS
LIN {X -133.2857,Y 13.8089,Z 192,A 174.0118,B 0.3433,C -0.0024,E1 0.1845,E2 280.4402} C_DIS
LIN {X -133.2857,Y 13.8089,Z 192,A 174.0102,B 0.3433,C -0.0024,E1 0.1845,E2 280.442} C_DIS
LIN {X -133.5618,Y 10.8147,Z 192,A 176.2831,B 0.3433,C 0.0035,E1 0.184,E2 278.0546} C_DIS
LIN {X -133.5618,Y 10.8147,Z 192,A 176.2818,B 0.3433,C 0.0035,E1 0.184,E2 278.056} C_DIS
LIN {X -133.8024,Y 7.2608,Z 192,A 178.8639,B 0.3432,C 0.0102,E1 0.1835,E2 275.3488} C_DIS
LIN {X -133.8024,Y 7.2608,Z 192,A 178.8625,B 0.3432,C 0.0102,E1 0.1835,E2 275.3503} C_DIS
LIN {X -133.9319,Y 4.2488,Z 192,A -178.6664,B 0.3429,C 0.0167,E1 0.1832,E2 272.7363} C_DIS
LIN {X -133.9319,Y 4.2488,Z 192,A -178.6681,B 0.3429,C 0.0167,E1 0.1832,E2 272.7382} C_DIS
LIN {X -133.9998,Y 0.3539,Z 192,A -175.571,B 0.3424,C 0.0247,E1 0.1832,E2 269.464} C_DIS
LIN {X -133.9998,Y 0.3539,Z 192,A -175.5737,B 0.3424,C 0.0247,E1 0.1832,E2 269.467} C_DIS
LIN {X -133.9585,Y -3.289,Z 192,A -172.9526,B 0.3419,C 0.0316,E1 0.1832,E2 266.7117} C_DIS
LIN {X -133.9585,Y -3.289,Z 192,A -172.9541,B 0.3419,C 0.0316,E1 0.1832,E2 266.7133} C_DIS
LIN {X -133.8369,Y -6.5731,Z 192,A -170.4827,B 0.3412,C 0.038,E1 0.1836,E2 264.1049} C_DIS
LIN {X -133.8369,Y -6.5731,Z 192,A -170.4842,B 0.3412,C 0.038,E1 0.1836,E2 264.1065} C_DIS
LIN {X -133.6354,Y -9.8534,Z 192,A -168.0186,B 0.3404,C 0.0443,E1 0.1841,E2 261.5023} C_DIS
LIN {X -133.6354,Y -9.8534,Z 192,A -168.0199,B 0.3404,C 0.0443,E1 0.1841,E2 261.5039} C_DIS
LIN {X -133.353,Y -13.1371,Z 192,A -165.5558,B 0.3396,C 0.0506,E1 0.1848,E2 258.8996} C_DIS
LIN {X -133.353,Y -13.1371,Z 192,A -165.5571,B 0.3396,C 0.0506,E1 0.1848,E2 258.9012} C_DIS
LIN {X -132.9533,Y -16.7153,Z 192,A -162.9395,B 0.3385,C 0.0572,E1 0.1857,E2 256.1384} C_DIS
LIN {X -132.9533,Y -16.7153,Z 192,A -162.9408,B 0.3385,C 0.0572,E1 0.1857,E2 256.1399} C_DIS
LIN {X -132.5498,Y -19.6601,Z 192,A -160.6796,B 0.3375,C 0.0628,E1 0.1866,E2 253.7432} C_DIS
LIN {X -132.5498,Y -19.6601,Z 192,A -160.6808,B 0.3375,C 0.0628,E1 0.1866,E2 253.7446} C_DIS
LIN {X -132.0279,Y -22.9042,Z 192,A -158.232,B 0.3363,C 0.0688,E1 0.1878,E2 251.1512} C_DIS
LIN {X -132.0279,Y -22.9042,Z 192,A -158.2332,B 0.3363,C 0.0688,E1 0.1878,E2 251.1526} C_DIS
LIN {X -131.2881,Y -26.8122,Z 192,A -155.3652,B 0.3349,C 0.0757,E1 0.1895,E2 248.1206} C_DIS
LIN {X -131.2881,Y -26.8122,Z 192,A -155.3666,B 0.3349,C 0.0757,E1 0.1895,E2 248.1223} C_DIS
LIN {X -130.5285,Y -30.2978,Z 192,A -152.5742,B 0.3333,C 0.0822,E1 0.1913,E2 245.1493} C_DIS
LIN {X -130.5285,Y -30.2978,Z 192,A -152.5761,B 0.3333,C 0.0822,E1 0.1913,E2 245.1515} C_DIS
LIN {X -129.3893,Y -34.8415,Z 192,A -149.2859,B 0.3314,C 0.0897,E1 0.1938,E2 241.6755} C_DIS
LIN {X -129.3893,Y -34.8415,Z 192,A -149.2876,B 0.3314,C 0.0897,E1 0.1938,E2 241.6775} C_DIS
LIN {X -128.0359,Y -39.5262,Z 192,A -146.1275,B 0.3294,C 0.0967,E1 0.1965,E2 238.3605} C_DIS
LIN {X -128.0359,Y -39.5262,Z 192,A -146.1286,B 0.3294,C 0.0967,E1 0.1965,E2 238.3618} C_DIS
LIN {X -127.0426,Y -42.6105,Z 192,A -143.8781,B 0.328,C 0.1015,E1 0.1987,E2 235.9836} C_DIS
LIN {X -125.6693,Y -46.507,Z 192,A -141.0632,B 0.3261,C 0.1073,E1 0.2016,E2 233.0129} C_DIS
LIN {X -125.6693,Y -46.507,Z 192,A -141.0642,B 0.3261,C 0.1073,E1 0.2016,E2 233.014} C_DIS
LIN {X -124.4181,Y -49.7561,Z 192,A -138.8607,B 0.3246,C 0.1117,E1 0.2041,E2 230.7034} C_DIS
LIN {X -123.1607,Y -52.7919,Z 192,A -136.7336,B 0.3232,C 0.1158,E1 0.2066,E2 228.4674} C_DIS
LIN {X -121.8296,Y -55.7957,Z 192,A -134.6013,B 0.3217,C 0.1198,E1 0.2093,E2 226.2248} C_DIS
LIN {X -120.4203,Y -58.7762,Z 192,A -132.5752,B 0.3204,C 0.1234,E1 0.212,E2 224.1047} C_DIS
LIN {X -118.8021,Y -61.9802,Z 192,A -130.3255,B 0.3189,C 0.1272,E1 0.2152,E2 221.7455} C_DIS
LIN {X -117.0586,Y -65.2175,Z 192,A -128.1215,B 0.3174,C 0.1308,E1 0.2185,E2 219.4444} C_DIS
LIN {X -115.2844,Y -68.3047,Z 192,A -125.8236,B 0.316,C 0.1343,E1 0.2222,E2 217.0264} C_DIS
LIN {X -112.8479,Y -72.2583,Z 192,A -123.3081,B 0.3143,C 0.138,E1 0.2264,E2 214.4288} C_DIS
LIN {X -111.0447,Y -75,Z 192,A -121.2551,B 0.3131,C 0.1408,E1 0.23,E2 212.2744} C_DIS
LIN {X -108.601,Y -78.4968,Z 192,A -119.0191,B 0.3118,C 0.1437,E1 0.2341,E2 209.974} C_DIS
LIN {X -106.1437,Y -81.7898,Z 192,A -116.6968,B 0.3105,C 0.1464,E1 0.2385,E2 207.563} C_DIS
LIN {X -103.5825,Y -85.0097,Z 192,A -114.465,B 0.3093,C 0.1489,E1 0.243,E2 205.2568} C_DIS
LIN {X -100.7047,Y -88.4003,Z 192,A -112.1149,B 0.3082,C 0.1512,E1 0.2478,E2 202.8358} C_DIS
LIN {X -97.9479,Y -91.4447,Z 192,A -109.9794,B 0.3072,C 0.1532,E1 0.2524,E2 200.6403} C_DIS
LIN {X -94.7645,Y -94.7405,Z 192,A -107.6886,B 0.3063,C 0.1551,E1 0.2576,E2 198.2968} C_DIS
LIN {X -91.8384,Y -97.5789,Z 192,A -105.7057,B 0.3056,C 0.1565,E1 0.2621,E2 196.2756} C_DIS
LIN {X -88.7638,Y -100.3837,Z 192,A -103.676,B 0.3049,C 0.1578,E1 0.2669,E2 194.2058} C_DIS
LIN {X -85.3765,Y -103.2801,Z 192,A -101.5504,B 0.3043,C 0.159,E1 0.2721,E2 192.0449} C_DIS
LIN {X -82.0833,Y -105.9162,Z 192,A -99.6119,B 0.3038,C 0.1599,E1 0.2769,E2 190.0845} C_DIS
LIN {X -79.275,Y -108.0342,Z 192,A -97.9835,B 0.3035,C 0.1606,E1 0.2811,E2 188.4359} C_DIS
LIN {X -75.8009,Y -110.4995,Z 192,A -96.0958,B 0.3031,C 0.1612,E1 0.286,E2 186.5371} C_DIS
LIN {X -73.0722,Y -112.3227,Z 192,A -94.6278,B 0.3029,C 0.1615,E1 0.2899,E2 185.0583} C_DIS
LIN {X -69.7226,Y -114.4326,Z 192,A -92.8689,B 0.3028,C 0.1618,E1 0.2946,E2 183.2882} C_DIS
LIN {X -66.6616,Y -116.2421,Z 192,A -91.1955,B 0.3028,C 0.1619,E1 0.2993,E2 181.5898} C_DIS
LIN {X -63.1684,Y -118.1768,Z 192,A -89.437,B 0.3028,C 0.1619,E1 0.3042,E2 179.8225} C_DIS
LIN {X -59.6353,Y -119.9964,Z 192,A -87.8543,B 0.3028,C 0.1619,E1 0.3086,E2 178.2576} C_DIS
LIN {X -56.3838,Y -121.5576,Z 192,A -86.492,B 0.3028,C 0.1619,E1 0.3124,E2 176.9234} C_DIS
LIN {X -53.6769,Y -122.7781,Z 192,A -85.1765,B 0.3028,C 0.1617,E1 0.3162,E2 175.5999} C_DIS
LIN {X -50.6569,Y -124.0549,Z 192,A -83.7538,B 0.3031,C 0.1613,E1 0.3203,E2 174.1731} C_DIS
LIN {X -47.3443,Y -125.3557,Z 192,A -82.4658,B 0.3031,C 0.1611,E1 0.324,E2 172.9217} C_DIS
LIN {X -44.5303,Y -126.3839,Z 192,A -81.096,B 0.3035,C 0.1605,E1 0.3281,E2 171.537} C_DIS
LIN {X -40.4698,Y -127.7408,Z 192,A -79.4624,B 0.3038,C 0.1599,E1 0.3329,E2 169.9337} C_DIS
LIN {X -37.3192,Y -128.6966,Z 192,A -78.1643,B 0.3041,C 0.1594,E1 0.3368,E2 168.6522} C_DIS
LIN {X -34.1516,Y -129.5733,Z 192,A -76.7728,B 0.3045,C 0.1586,E1 0.341,E2 167.2622} C_DIS
LIN {X -30.2996,Y -130.5281,Z 192,A -75.2767,B 0.3049,C 0.1578,E1 0.3454,E2 165.7969} C_DIS
LIN {X -26.1432,Y -131.4242,Z 192,A -73.7145,B 0.3054,C 0.1569,E1 0.3501,E2 164.2744} C_DIS
LIN {X -22.5624,Y -132.0858,Z 192,A -72.4213,B 0.3058,C 0.1561,E1 0.3539,E2 163.0222} C_DIS
LIN {X -19.6629,Y -132.5494,Z 192,A -71.1547,B 0.3063,C 0.1551,E1 0.3579,E2 161.7529} C_DIS
LIN {X -15.7344,Y -133.0711,Z 192,A -69.7102,B 0.3068,C 0.154,E1 0.3622,E2 160.3469} C_DIS
LIN {X -12.1975,Y -133.4432,Z 192,A -68.4367,B 0.3073,C 0.153,E1 0.366,E2 159.1117} C_DIS
LIN {X -9.2045,Y -133.6828,Z 192,A -67.1954,B 0.3079,C 0.1518,E1 0.3698,E2 157.8762} C_DIS
LIN {X -5.894,Y -133.8702,Z 192,A -66.0465,B 0.3084,C 0.1508,E1 0.3733,E2 156.7689} C_DIS
LIN {X -1.6558,Y -133.9892,Z 192,A -64.5696,B 0.3091,C 0.1495,E1 0.3776,E2 155.344} C_DIS
LIN {X 0.9701,Y -133.9923,Z 192,A -63.8182,B 0.3093,C 0.149,E1 0.3798,E2 154.6506} C_DIS
Enddeposition()
LIN {X 0.9701,Y -133.9923,Z 192,A -63.8185,B 0.3093,C 0.149,E1 0.3798,E2 154.6509} C_DIS
Startdeposition()
$VEL.CP = VEL_PRINT
LIN {X -1.9561,Y -134.8833,Z 192,A -65.2194,B 0.3083,C 0.1508,E1 0.3752,E2 156.0861} C_DIS
LIN {X -6.3855,Y -134.7464,Z 192,A -66.9936,B 0.3074,C 0.1527,E1 0.3698,E2 157.8445} C_DIS
LIN {X -9.603,Y -134.555,Z 192,A -67.9787,B 0.3071,C 0.1533,E1 0.3669,E2 158.7693} C_DIS
LIN {X -12.7587,Y -134.2924,Z 192,A -69.1321,B 0.3066,C 0.1542,E1 0.3635,E2 159.8931} C_DIS
LIN {X -16.4726,Y -133.8884,Z 192,A -70.4736,B 0.3061,C 0.1552,E1 0.3594,E2 161.1965} C_DIS
LIN {X -19.4703,Y -133.485,Z 192,A -71.7159,B 0.3056,C 0.1563,E1 0.3556,E2 162.4329} C_DIS
LIN {X -23.8172,Y -132.7777,Z 192,A -73.2287,B 0.3051,C 0.1571,E1 0.3512,E2 163.8897} C_DIS
LIN {X -27.0946,Y -132.148,Z 192,A -74.5433,B 0.3047,C 0.158,E1 0.3472,E2 165.1887} C_DIS
LIN {X -31.0149,Y -131.2844,Z 192,A -76.16,B 0.3041,C 0.159,E1 0.3423,E2 166.7924} C_DIS
LIN {X -34.8093,Y -130.3283,Z 192,A -77.6049,B 0.3038,C 0.1597,E1 0.338,E2 168.2036} C_DIS
LIN {X -38.4822,Y -129.2927,Z 192,A -79.0571,B 0.3035,C 0.1603,E1 0.3337,E2 169.6297} C_DIS
LIN {X -41.9109,Y -128.223,Z 192,A -80.6055,B 0.3031,C 0.1611,E1 0.329,E2 171.1826} C_DIS
LIN {X -47.3536,Y -126.3121,Z 192,A -82.5052,B 0.3029,C 0.1613,E1 0.3237,E2 172.9953} C_DIS
LIN {X -50.2296,Y -125.1964,Z 192,A -84.1168,B 0.3025,C 0.1621,E1 0.3188,E2 174.6561} C_DIS
LIN {X -53.9926,Y -123.621,Z 192,A -85.7402,B 0.3024,C 0.1623,E1 0.3141,E2 176.2628} C_DIS
LIN {X -57.4419,Y -122.0579,Z 192,A -87.2784,B 0.3023,C 0.1625,E1 0.3098,E2 177.7905} C_DIS
LIN {X -61.4917,Y -120.0664,Z 192,A -89.1979,B 0.3023,C 0.1626,E1 0.3043,E2 179.7113} C_DIS
LIN {X -64.7402,Y -118.3485,Z 192,A -91.0019,B 0.3021,C 0.1628,E1 0.2992,E2 181.5549} C_DIS
LIN {X -69.2916,Y -115.7427,Z 192,A -93.1398,B 0.3023,C 0.1624,E1 0.2934,E2 183.6794} C_DIS
LIN {X -72.8322,Y -113.5478,Z 192,A -94.9438,B 0.3025,C 0.162,E1 0.2886,E2 185.4895} C_DIS
LIN {X -76.7438,Y -110.9421,Z 192,A -96.968,B 0.3029,C 0.1614,E1 0.2833,E2 187.5189} C_DIS
LIN {X -80.0359,Y -108.5906,Z 192,A -98.9359,B 0.3032,C 0.1608,E1 0.2782,E2 189.5272} C_DIS
LIN {X -85.327,Y -104.4841,Z 192,A -101.8887,B 0.304,C 0.1593,E1 0.2709,E2 192.498} C_DIS
LIN {X -88.2775,Y -102.004,Z 192,A -103.8696,B 0.3045,C 0.1583,E1 0.266,E2 194.5342} C_DIS
LIN {X -93.458,Y -97.2797,Z 192,A -107.7779,B 0.3057,C 0.1559,E1 0.2568,E2 198.5912} C_DIS
LIN {X -96.6193,Y -94.141,Z 192,A -109.2146,B 0.3066,C 0.1543,E1 0.2538,E2 199.9557} C_DIS
LIN {X -99.7289,Y -90.8396,Z 192,A -111.8391,B 0.3077,C 0.1521,E1 0.248,E2 202.6914} C_DIS
LIN {X -102.6292,Y -87.5495,Z 192,A -114.1426,B 0.3088,C 0.1498,E1 0.2432,E2 205.0648} C_DIS
LIN {X -106.0133,Y -83.4196,Z 192,A -116.9779,B 0.3103,C 0.1467,E1 0.2376,E2 207.9899} C_DIS
LIN {X -108.8034,Y -79.7463,Z 192,A -119.4927,B 0.3117,C 0.1436,E1 0.2328,E2 210.5922} C_DIS
LIN {X -111.4553,Y -75.9968,Z 192,A -122.1043,B 0.3132,C 0.1402,E1 0.2281,E2 213.3074} C_DIS
LIN {X -113.708,Y -72.5821,Z 192,A -124.3269,B 0.3146,C 0.137,E1 0.2243,E2 215.6058} C_DIS
LIN {X -115.7139,Y -69.3398,Z 192,A -126.5827,B 0.3161,C 0.1337,E1 0.2206,E2 217.9607} C_DIS
LIN {X -117.6277,Y -66.0405,Z 192,A -128.8081,B 0.3176,C 0.1302,E1 0.2172,E2 220.2799} C_DIS
LIN {X -119.6992,Y -62.2052,Z 192,A -131.3547,B 0.3193,C 0.1259,E1 0.2135,E2 222.9337} C_DIS
LIN {X -121.0142,Y -59.604,Z 192,A -133.1794,B 0.3205,C 0.1227,E1 0.211,E2 224.8485} C_DIS
LIN {X -122.4241,Y -56.6517,Z 192,A -135.2606,B 0.3219,C 0.119,E1 0.2082,E2 227.0354} C_DIS
LIN {X -123.9101,Y -53.3237,Z 192,A -137.6296,B 0.3235,C 0.1145,E1 0.2053,E2 229.529} C_DIS
LIN {X -125.2321,Y -50.141,Z 192,A -139.8534,B 0.325,C 0.1102,E1 0.2027,E2 231.8675} C_DIS
LIN {X -127.3489,Y -44.4913,Z 192,A -144.5397,B 0.3281,C 0.1008,E1 0.1978,E2 236.8707} C_DIS
LIN {X -128.6629,Y -40.5372,Z 192,A -146.6081,B 0.3295,C 0.0961,E1 0.1959,E2 238.9825} C_DIS
LIN {X -129.6218,Y -37.3583,Z 192,A -149.3976,B 0.3312,C 0.0901,E1 0.1935,E2 241.9737} C_DIS
LIN {X -130.4846,Y -34.2231,Z 192,A -151.1257,B 0.3323,C 0.086,E1 0.1922,E2 243.7516} C_DIS
LIN {X -131.1905,Y -31.4047,Z 192,A -153.1454,B 0.3334,C 0.0813,E1 0.1907,E2 245.8841} C_DIS
LIN {X -131.8999,Y -28.2776,Z 192,A -155.5457,B 0.3347,C 0.0757,E1 0.1892,E2 248.4323} C_DIS
LIN {X -131.8999,Y -28.2776,Z 192,A -155.5469,B 0.3347,C 0.0757,E1 0.1892,E2 248.4336} C_DIS
LIN {X -132.562,Y -24.9919,Z 192,A -157.9852,B 0.336,C 0.0698,E1 0.1878,E2 251.0145} C_DIS
LIN {X -132.562,Y -24.9919,Z 192,A -157.9873,B 0.336,C 0.0698,E1 0.1878,E2 251.0169} C_DIS
LIN {X -133.2676,Y -20.9046,Z 192,A -161.0074,B 0.3375,C 0.0624,E1 0.1863,E2 254.2112} C_DIS
LIN {X -133.2676,Y -20.9046,Z 192,A -161.0092,B 0.3375,C 0.0624,E1 0.1863,E2 254.2133} C_DIS
LIN {X -133.8321,Y -16.9272,Z 192,A -164.1388,B 0.3388,C 0.0546,E1 0.1851,E2 257.5365} C_DIS
LIN {X -133.8321,Y -16.9272,Z 192,A -164.1414,B 0.3388,C 0.0546,E1 0.1851,E2 257.5395} C_DIS
LIN {X -134.3013,Y -12.6656,Z 192,A -167.1182,B 0.34,C 0.047,E1 0.1842,E2 260.6704} C_DIS
LIN {X -134.3013,Y -12.6656,Z 192,A -167.1198,B 0.34,C 0.047,E1 0.1842,E2 260.6723} C_DIS
LIN {X -134.6368,Y -8.3762,Z 192,A -170.2923,B 0.341,C 0.0388,E1 0.1835,E2 264.0209} C_DIS
LIN {X -134.6368,Y -8.3762,Z 192,A -170.2944,B 0.341,C 0.0388,E1 0.1835,E2 264.0233} C_DIS
LIN {X -134.8125,Y -4.8001,Z 192,A -173.0704,B 0.3417,C 0.0317,E1 0.1832,E2 266.9605} C_DIS
LIN {X -134.8125,Y -4.8001,Z 192,A -173.0725,B 0.3417,C 0.0317,E1 0.1832,E2 266.9628} C_DIS
LIN {X -134.8954,Y -0.8482,Z 192,A -175.9408,B 0.3423,C 0.0241,E1 0.183,E2 269.9805} C_DIS
LIN {X -134.8954,Y -0.8482,Z 192,A -175.9425,B 0.3423,C 0.0241,E1 0.183,E2 269.9825} C_DIS
LIN {X -134.876,Y 2.3903,Z 192,A -178.5464,B 0.3428,C 0.0174,E1 0.1831,E2 272.7376} C_DIS
LIN {X -134.876,Y 2.3903,Z 192,A -178.5484,B 0.3428,C 0.0174,E1 0.1831,E2 272.7399} C_DIS
LIN {X -134.7311,Y 6.6897,Z 192,A 178.2783,B 0.3431,C 0.009,E1 0.1835,E2 276.0748} C_DIS
LIN {X -134.7311,Y 6.6897,Z 192,A 178.2761,B 0.3431,C 0.009,E1 0.1835,E2 276.0773} C_DIS
LIN {X -134.4792,Y 10.6336,Z 192,A 175.1411,B 0.3431,C 0.0009,E1 0.1842,E2 279.3827} C_DIS
LIN {X -134.4792,Y 10.6336,Z 192,A 175.1381,B 0.3431,C 0.0009,E1 0.1842,E2 279.3861} C_DIS
LIN {X -134.1252,Y 14.4091,Z 192,A 172.4475,B 0.3431,C -0.0061,E1 0.185,E2 282.1994} C_DIS
LIN {X -134.1252,Y 14.4091,Z 192,A 172.4458,B 0.3431,C -0.0061,E1 0.185,E2 282.2013} C_DIS
LIN {X -133.6226,Y 18.5074,Z 192,A 169.2428,B 0.3429,C -0.0143,E1 0.1862,E2 285.565} C_DIS
LIN {X -133.6226,Y 18.5074,Z 192,A 169.24,B 0.3429,C -0.0143,E1 0.1862,E2 285.5681} C_DIS
LIN {X -133.038,Y 22.3175,Z 192,A 166.5787,B 0.3425,C -0.0211,E1 0.1874,E2 288.3395} C_DIS
LIN {X -133.038,Y 22.3175,Z 192,A 166.5772,B 0.3425,C -0.0211,E1 0.1874,E2 288.3411} C_DIS
LIN {X -132.3607,Y 26.0448,Z 192,A 163.7184,B 0.342,C -0.0283,E1 0.189,E2 291.331} C_DIS
LIN {X -132.3607,Y 26.0448,Z 192,A 163.7164,B 0.342,C -0.0283,E1 0.189,E2 291.3334} C_DIS
LIN {X -130.8132,Y 32.9411,Z 192,A 158.6022,B 0.3408,C -0.0408,E1 0.1924,E2 296.6598} C_DIS
LIN {X -130.8132,Y 32.9411,Z 192,A 158.5993,B 0.3408,C -0.0408,E1 0.1924,E2 296.663} C_DIS
LIN {X -129.8113,Y 36.6919,Z 192,A 155.843,B 0.3399,C -0.0474,E1 0.1946,E2 299.5259} C_DIS
LIN {X -129.8113,Y 36.6919,Z 192,A 155.8413,B 0.3399,C -0.0474,E1 0.1946,E2 299.5278} C_DIS
LIN {X -128.5827,Y 40.7883,Z 192,A 152.8529,B 0.3389,C -0.0543,E1 0.1972,E2 302.6253} C_DIS
LIN {X -128.5827,Y 40.7883,Z 192,A 152.8513,B 0.3389,C -0.0543,E1 0.1972,E2 302.6271} C_DIS
LIN {X -127.3146,Y 44.5902,Z 192,A 150.2695,B 0.3379,C -0.0601,E1 0.1997,E2 305.2883} C_DIS
LIN {X -127.3146,Y 44.5902,Z 192,A 150.2685,B 0.3379,C -0.0601,E1 0.1997,E2 305.2893} C_DIS
LIN {X -126.1931,Y 47.6713,Z 192,A 147.9981,B 0.337,C -0.065,E1 0.2021,E2 307.637} C_DIS
LIN {X -126.1931,Y 47.6713,Z 192,A 147.9972,B 0.337,C -0.065,E1 0.2021,E2 307.638} C_DIS
LIN {X -124.9105,Y 50.9387,Z 192,A 145.7175,B 0.336,C -0.0699,E1 0.2046,E2 309.9853} C_DIS
LIN {X -123.3418,Y 54.6271,Z 192,A 142.7467,B 0.3347,C -0.0759,E1 0.2082,E2 313.0615} C_DIS
LIN {X -123.3418,Y 54.6271,Z 192,A 142.7449,B 0.3347,C -0.0759,E1 0.2082,E2 313.0635} C_DIS
LIN {X -121.582,Y 58.4379,Z 192,A 140.3908,B 0.3336,C -0.0806,E1 0.2112,E2 315.463} C_DIS
LIN {X -119.86,Y 61.8973,Z 192,A 137.8546,B 0.3324,C -0.0853,E1 0.2147,E2 318.0693} C_DIS
LIN {X -117.7796,Y 65.7704,Z 192,A 135.2098,B 0.3312,C -0.09,E1 0.2186,E2 320.7731} C_DIS
LIN {X -115.7921,Y 69.2088,Z 192,A 133.0269,B 0.3301,C -0.0938,E1 0.222,E2 322.9924} C_DIS
LIN {X -114.2114,Y 71.7875,Z 192,A 130.901,B 0.3292,C -0.0971,E1 0.2254,E2 325.1793} C_DIS
LIN {X -111.6406,Y 75.7234,Z 192,A 128.3012,B 0.328,C -0.1011,E1 0.2299,E2 327.8211} C_DIS
LIN {X -109.161,Y 79.2559,Z 192,A 125.7718,B 0.3268,C -0.1047,E1 0.2344,E2 330.3978} C_DIS
LIN {X -106.6464,Y 82.6085,Z 192,A 123.4962,B 0.3259,C -0.1077,E1 0.2387,E2 332.7062} C_DIS
LIN {X -104.0245,Y 85.8869,Z 192,A 121.1683,B 0.3249,C -0.1106,E1 0.2433,E2 335.0693} C_DIS
LIN {X -100.8571,Y 89.5855,Z 192,A 118.7268,B 0.3239,C -0.1133,E1 0.2483,E2 337.534} C_DIS
LIN {X -98.1272,Y 92.5671,Z 192,A 116.5209,B 0.3232,C -0.1155,E1 0.253,E2 339.7703} C_DIS
LIN {X -94.9236,Y 95.8498,Z 192,A 114.0815,B 0.3224,C -0.1177,E1 0.2584,E2 342.2394} C_DIS
LIN {X -91.4913,Y 99.1315,Z 192,A 112.1582,B 0.3218,C -0.1194,E1 0.2628,E2 344.1559} C_DIS
LIN {X -89.3622,Y 101.0545,Z 192,A 110.4863,B 0.3213,C -0.1205,E1 0.2667,E2 345.8551} C_DIS
LIN {X -86.1503,Y 103.8064,Z 192,A 108.4434,B 0.3209,C -0.1218,E1 0.2717,E2 347.9119} C_DIS
LIN {X -82.7354,Y 106.5481,Z 192,A 106.1232,B 0.3204,C -0.123,E1 0.2775,E2 350.2585} C_DIS
LIN {X -80.0537,Y 108.5775,Z 192,A 105.1289,B 0.3202,C -0.1236,E1 0.2799,E2 351.2265} C_DIS
LIN {X -77.6322,Y 110.3217,Z 192,A 103.5314,B 0.32,C -0.1241,E1 0.284,E2 352.843} C_DIS
LIN {X -74.2261,Y 112.6415,Z 192,A 101.3443,B 0.3198,C -0.1247,E1 0.2898,E2 355.0548} C_DIS
LIN {X -71.2952,Y 114.5191,Z 192,A 100.3812,B 0.3196,C -0.125,E1 0.2923,E2 355.9871} C_DIS
LIN {X -68.9756,Y 115.9311,Z 192,A 98.9106,B 0.3196,C -0.1252,E1 0.2964,E2 357.4758} C_DIS
LIN {X -64.8762,Y 118.2743,Z 192,A 97.1733,B 0.3195,C -0.1254,E1 0.3011,E2 359.1966} C_DIS
LIN {X -61.3447,Y 120.1413,Z 192,A 95.2229,B 0.3195,C -0.1254,E1 0.3066,E2 361.161} C_DIS
LIN {X -57.4094,Y 122.0734,Z 192,A 93.4416,B 0.3195,C -0.1252,E1 0.3116,E2 362.9369} C_DIS
LIN {X -53.3783,Y 123.8866,Z 192,A 91.542,B 0.3197,C -0.1248,E1 0.3171,E2 364.8368} C_DIS
LIN {X -50.2093,Y 125.2046,Z 192,A 90.1902,B 0.3198,C -0.1245,E1 0.321,E2 366.1818} C_DIS
LIN {X -46.7805,Y 126.5267,Z 192,A 88.7478,B 0.32,C -0.124,E1 0.3253,E2 367.6166} C_DIS
LIN {X -42.0104,Y 128.1899,Z 192,A 86.8533,B 0.3203,C -0.1233,E1 0.3309,E2 369.4953} C_DIS
LIN {X -37.6886,Y 129.5251,Z 192,A 85.0019,B 0.3207,C -0.1223,E1 0.3364,E2 371.3417} C_DIS
LIN {X -34.1192,Y 130.5123,Z 192,A 83.4694,B 0.321,C -0.1214,E1 0.341,E2 372.8711} C_DIS
LIN {X -30.2049,Y 131.4718,Z 192,A 81.9535,B 0.3214,C -0.1204,E1 0.3456,E2 374.3745} C_DIS
LIN {X -26.6222,Y 132.2441,Z 192,A 80.5847,B 0.3217,C -0.1195,E1 0.3498,E2 375.7312} C_DIS
LIN {X -20.3198,Y 133.3581,Z 192,A 78.3031,B 0.3224,C -0.1177,E1 0.3567,E2 377.9848} C_DIS
LIN {X -16.8668,Y 133.84,Z 192,A 76.8526,B 0.3229,C -0.1164,E1 0.3612,E2 379.4329} C_DIS
LIN {X -12.7265,Y 134.2954,Z 192,A 75.4045,B 0.3233,C -0.115,E1 0.3656,E2 380.86} C_DIS
LIN {X -8.0832,Y 134.6548,Z 192,A 73.7825,B 0.3239,C -0.1134,E1 0.3705,E2 382.4586} C_DIS
LIN {X -4.9877,Y 134.8051,Z 192,A 72.5037,B 0.3244,C -0.112,E1 0.3745,E2 383.7345} C_DIS
LIN {X -0.1586,Y 134.8984,Z 192,A 70.8356,B 0.325,C -0.1102,E1 0.3796,E2 385.377} C_DIS
LIN {X 3.9466,Y 134.8395,Z 192,A 69.3655,B 0.3256,C -0.1084,E1 0.384,E2 386.8284} C_DIS
LIN {X 8.3438,Y 134.6388,Z 192,A 67.9394,B 0.3262,C -0.1067,E1 0.3883,E2 388.2241} C_DIS
LIN {X 12.5095,Y 134.3163,Z 192,A 66.509,B 0.3268,C -0.1048,E1 0.3926,E2 389.6305} C_DIS
LIN {X 16.1989,Y 133.921,Z 192,A 65.3139,B 0.3273,C -0.1033,E1 0.3961,E2 390.7988} C_DIS
LIN {X 19.3472,Y 133.5026,Z 192,A 64.1476,B 0.3278,C -0.1016,E1 0.3996,E2 391.9518} C_DIS
LIN {X 23.8829,Y 132.7659,Z 192,A 62.6397,B 0.3285,C -0.0995,E1 0.404,E2 393.4277} C_DIS
LIN {X 27.0392,Y 132.1592,Z 192,A 61.5609,B 0.3289,C -0.0979,E1 0.4072,E2 394.4855} C_DIS
LIN {X 30.6376,Y 131.373,Z 192,A 60.317,B 0.3295,C -0.096,E1 0.4108,E2 395.7057} C_DIS
LIN {X 33.7837,Y 130.5993,Z 192,A 59.2182,B 0.33,C -0.0943,E1 0.4139,E2 396.7837} C_DIS
LIN {X 36.4143,Y 129.889,Z 192,A 58.3083,B 0.3304,C -0.0928,E1 0.4165,E2 397.6748} C_DIS
LIN {X 39.6054,Y 128.9518,Z 192,A 57.2452,B 0.3309,C -0.0911,E1 0.4195,E2 398.7113} C_DIS
LIN {X 44.9302,Y 127.1967,Z 192,A 55.3603,B 0.3317,C -0.0879,E1 0.4247,E2 400.5579} C_DIS
LIN {X 49.0746,Y 125.6536,Z 192,A 53.8636,B 0.3324,C -0.0853,E1 0.4288,E2 402.0244} C_DIS
LIN {X 52.4835,Y 124.2693,Z 192,A 52.6547,B 0.333,C -0.0832,E1 0.4321,E2 403.2052} C_DIS
LIN {X 55.6378,Y 122.8898,Z 192,A 51.5854,B 0.3334,C -0.0813,E1 0.4349,E2 404.243} C_DIS
LIN {X 58.424,Y 121.5887,Z 192,A 50.5676,B 0.3339,C -0.0794,E1 0.4375,E2 405.2372} C_DIS
LIN {X 61.8373,Y 119.8905,Z 192,A 49.0033,B 0.3346,C -0.0762,E1 0.4416,E2 406.7969} C_DIS
LIN {X 65.5118,Y 117.9231,Z 192,A 48.1573,B 0.3349,C -0.075,E1 0.4436,E2 407.5663} C_DIS
LIN {X 65.5118,Y 117.9231,Z 192,A 48.1563,B 0.3349,C -0.075,E1 0.4436,E2 407.5674} C_DIS
LIN {X 69.5799,Y 115.5696,Z 192,A 46.4682,B 0.3356,C -0.0716,E1 0.4478,E2 409.2293} C_DIS
LIN {X 73.485,Y 113.1264,Z 192,A 45.2002,B 0.3361,C -0.0693,E1 0.4508,E2 410.4381} C_DIS
LIN {X 76.0031,Y 111.4509,Z 192,A 43.996,B 0.3367,C -0.0667,E1 0.4537,E2 411.6353} C_DIS
LIN {X 79.6819,Y 108.8507,Z 192,A 42.6011,B 0.3372,C -0.0639,E1 0.4569,E2 412.9846} C_DIS
LIN {X 83.0485,Y 106.3048,Z 192,A 41.2379,B 0.3377,C -0.0611,E1 0.46,E2 414.3096} C_DIS
LIN {X 86.4753,Y 103.5361,Z 192,A 39.873,B 0.3382,C -0.0583,E1 0.4629,E2 415.6287} C_DIS
LIN {X 89.7567,Y 100.7048,Z 192,A 38.4964,B 0.3387,C -0.0554,E1 0.4658,E2 416.9628} C_DIS
LIN {X 92.9776,Y 97.7389,Z 192,A 37.3073,B 0.3391,C -0.053,E1 0.4682,E2 418.0895} C_DIS
LIN {X 95.3725,Y 95.4038,Z 192,A 36.0916,B 0.3395,C -0.0502,E1 0.4706,E2 419.2859} C_DIS
LIN {X 98.5055,Y 92.165,Z 192,A 34.6848,B 0.3399,C -0.0472,E1 0.4733,E2 420.6444} C_DIS
LIN {X 101.485,Y 88.8734,Z 192,A 33.3223,B 0.3403,C -0.0442,E1 0.4758,E2 421.9565} C_DIS
LIN {X 104.2934,Y 85.5604,Z 192,A 31.9705,B 0.3407,C -0.0412,E1 0.4782,E2 423.2601} C_DIS
LIN {X 107.2041,Y 81.8836,Z 192,A 30.5327,B 0.3411,C -0.038,E1 0.4806,E2 424.643} C_DIS
LIN {X 109.743,Y 78.448,Z 192,A 29.0082,B 0.3415,C -0.0343,E1 0.4831,E2 426.1386} C_DIS
LIN {X 111.9357,Y 75.2874,Z 192,A 28.0541,B 0.3417,C -0.0324,E1 0.4846,E2 427.0238} C_DIS
LIN {X 114.2094,Y 71.7907,Z 192,A 26.7588,B 0.3419,C -0.0295,E1 0.4865,E2 428.2702} C_DIS
LIN {X 116.7559,Y 67.5699,Z 192,A 25.3701,B 0.3422,C -0.0265,E1 0.4884,E2 429.5853} C_DIS
LIN {X 118.5495,Y 64.3717,Z 192,A 24.1145,B 0.3424,C -0.0234,E1 0.49,E2 430.8091} C_DIS
LIN {X 120.3228,Y 60.9882,Z 192,A 22.9884,B 0.3426,C -0.0208,E1 0.4914,E2 431.8823} C_DIS
LIN {X 122.5229,Y 56.4382,Z 192,A 21.4519,B 0.3428,C -0.0173,E1 0.4932,E2 433.353} C_DIS
LIN {X 123.8961,Y 53.3563,Z 192,A 20.4479,B 0.3428,C -0.015,E1 0.4943,E2 434.3102} C_DIS
LIN {X 125.1491,Y 50.3469,Z 192,A 19.409,B 0.343,C -0.0125,E1 0.4954,E2 435.3111} C_DIS
LIN {X 127.0043,Y 45.4655,Z 192,A 17.8659,B 0.343,C -0.0089,E1 0.4968,E2 436.7791} C_DIS
LIN {X 128.1947,Y 41.9959,Z 192,A 16.7543,B 0.3431,C -0.0063,E1 0.4977,E2 437.8406} C_DIS
LIN {X 129.1225,Y 39.0473,Z 192,A 15.7398,B 0.3431,C -0.0038,E1 0.4986,E2 438.8213} C_DIS
LIN {X 130.2748,Y 35.0099,Z 192,A 14.5106,B 0.3431,C -0.001,E1 0.4994,E2 439.987} C_DIS
LIN {X 131.1862,Y 31.4225,Z 192,A 13.4063,B 0.3431,C 0.0016,E1 0.5001,E2 441.0372} C_DIS
LIN {X 131.9138,Y 28.2129,Z 192,A 12.3632,B 0.3431,C 0.0041,E1 0.5007,E2 442.0391} C_DIS
LIN {X 132.7762,Y 23.8255,Z 192,A 11.0154,B 0.3431,C 0.0073,E1 0.5014,E2 443.3221} C_DIS
LIN {X 133.3544,Y 20.3439,Z 192,A 9.9555,B 0.3431,C 0.0098,E1 0.5019,E2 444.3299} C_DIS
LIN {X 133.8077,Y 17.1131,Z 192,A 8.8603,B 0.343,C 0.0125,E1 0.5022,E2 445.3906} C_DIS
LIN {X 134.3621,Y 12.0198,Z 192,A 7.4416,B 0.3428,C 0.0156,E1 0.5026,E2 446.7177} C_DIS
LIN {X 134.6007,Y 8.9613,Z 192,A 6.3498,B 0.3428,C 0.0185,E1 0.5028,E2 447.7841} C_DIS
LIN {X 134.8055,Y 4.9776,Z 192,A 5.2507,B 0.3426,C 0.0209,E1 0.503,E2 448.8101} C_DIS
LIN {X 134.8995,Y 0.2096,Z 192,A 3.8524,B 0.3423,C 0.0241,E1 0.503,E2 450.1307} C_DIS
LIN {X 134.8659,Y -2.9961,Z 192,A 2.6172,B 0.3421,C 0.0274,E1 0.503,E2 451.3507} C_DIS
LIN {X 134.6508,Y -8.1481,Z 192,A 1.2373,B 0.3419,C 0.0304,E1 0.5028,E2 452.6283} C_DIS
LIN {X 134.3669,Y -11.9629,Z 192,A -0.1085,B 0.3415,C 0.0338,E1 0.5025,E2 453.9392} C_DIS
LIN {X 133.8936,Y -16.429,Z 192,A -1.2714,B 0.3413,C 0.0362,E1 0.5021,E2 455.0065} C_DIS
Enddeposition()
END
